Yaskawa INFORM job: DPRINT3D14.JBI

/JOB
//NAME DPRINT3D14
//POS
///NPOS 1103,0,0,0,0,0
///TOOL 9
///POSTYPE PULSE
///PULSE
C00000=35589,48234,-113777,79423,-119050,-86602,0
C00001=36149,47910,-114639,78756,-119195,-86909,0
C00002=39346,46465,-118547,75010,-120071,-88397,0
C00003=40415,47046,-117012,74132,-121018,-88120,0
C00004=36113,47361,-116093,78604,-118868,-87310,0
C00005=40186,44054,-125164,73265,-118809,-90339,0
C00006=40186,43993,-125176,73276,-118834,-90313,0
C00007=35105,44450,-123810,78705,-116693,-89341,0
C00008=36407,44998,-122328,77544,-117679,-89063,0
C00009=36336,47795,-114813,78560,-119287,-86953,0
C00010=40997,44020,-125117,72434,-119231,-90399,0
C00011=39991,43550,-126414,73325,-118416,-90634,0
C00012=35373,47318,-116057,79359,-118479,-87184,0
C00013=36258,47755,-114917,78624,-119220,-86972,0
C00014=35643,48123,-113935,79362,-119070,-86625,0
C00015=36516,48577,-112760,78655,-119824,-86406,0
C00016=42226,43977,-125263,71121,-119762,-90600,0
C00017=39858,42875,-128320,73230,-117847,-91152,0
C00018=34271,47458,-115667,80501,-117931,-86950,0
C00019=35173,47889,-114544,79748,-118673,-86739,0
C00020=34938,48134,-113895,80062,-118666,-86531,0
C00021=35406,48369,-113288,79679,-119063,-86417,0
C00022=35589,48179,-113789,79434,-119069,-86578,0
C00023=36149,47855,-114651,78767,-119213,-86885,0
C00024=39346,46408,-118558,75022,-120093,-88372,0
C00025=40382,46970,-117074,74172,-121010,-88104,0
C00026=36113,47305,-116105,78615,-118886,-87285,0
C00027=40186,43993,-125176,73276,-118834,-90313,0
C00028=40187,43932,-125189,73288,-118859,-90287,0
C00029=35144,44406,-123780,78681,-116742,-89307,0
C00030=36408,44938,-122340,77555,-117701,-89037,0
C00031=36336,47739,-114825,78571,-119305,-86929,0
C00032=40998,43959,-125128,72446,-119256,-90373,0
C00033=39991,43488,-126425,73337,-118441,-90607,0
C00034=35373,47262,-116069,79370,-118497,-87160,0
C00035=36259,47699,-114928,78635,-119239,-86948,0
C00036=35643,48068,-113947,79373,-119088,-86601,0
C00037=36517,48522,-112772,78666,-119842,-86382,0
C00038=42227,43916,-125274,71133,-119788,-90574,0
C00039=39859,42812,-128333,73241,-117873,-91125,0
C00040=34271,47402,-115679,80511,-117948,-86926,0
C00041=35173,47834,-114556,79759,-118692,-86714,0
C00042=34938,48079,-113907,80073,-118685,-86507,0
C00043=35406,48314,-113299,79690,-119081,-86392,0
C00044=35589,48124,-113800,79445,-119086,-86554,0
C00045=36150,47799,-114663,78778,-119233,-86861,0
C00046=39347,46350,-118571,75034,-120114,-88347,0
C00047=40348,46895,-117136,74211,-121001,-88089,0
C00048=36114,47249,-116118,78626,-118905,-87261,0
C00049=40187,43932,-125189,73288,-118859,-90287,0
C00050=40187,43871,-125200,73300,-118885,-90260,0
C00051=35183,44361,-123750,78656,-116791,-89272,0
C00052=36408,44879,-122352,77566,-117722,-89011,0
C00053=36337,47684,-114837,78583,-119324,-86904,0
C00054=40998,43898,-125141,72457,-119282,-90347,0
C00055=39992,43426,-126438,73348,-118466,-90581,0
C00056=35373,47206,-116081,79381,-118516,-87135,0
C00057=36259,47644,-114940,78647,-119258,-86923,0
C00058=35643,48013,-113959,79384,-119105,-86577,0
C00059=36517,48468,-112784,78678,-119860,-86358,0
C00060=42227,43855,-125287,71145,-119816,-90548,0
C00061=39859,42749,-128346,73252,-117899,-91098,0
C00062=34272,47346,-115691,80521,-117965,-86901,0
C00063=35174,47778,-114567,79770,-118709,-86690,0
C00064=34938,48024,-113919,80084,-118702,-86482,0
C00065=35407,48259,-113311,79701,-119098,-86369,0
C00066=35589,48069,-113812,79456,-119104,-86529,0
C00067=36150,47744,-114675,78789,-119251,-86836,0
C00068=39347,46293,-118583,75046,-120136,-88322,0
C00069=40315,46819,-117198,74251,-120993,-88073,0
C00070=36114,47193,-116129,78637,-118924,-87236,0
C00071=40187,43871,-125200,73300,-118885,-90260,0
C00072=40188,43810,-125213,73311,-118909,-90234,0
C00073=35222,44317,-123719,78632,-116840,-89237,0
C00074=36408,44820,-122364,77576,-117742,-88985,0
C00075=36337,47628,-114848,78594,-119343,-86880,0
C00076=40999,43837,-125153,72469,-119308,-90321,0
C00077=39992,43364,-126451,73360,-118492,-90554,0
C00078=35374,47150,-116092,79391,-118534,-87111,0
C00079=36259,47588,-114951,78658,-119277,-86899,0
C00080=35644,47958,-113971,79395,-119124,-86553,0
C00081=36517,48413,-112796,78689,-119879,-86334,0
C00082=42228,43794,-125299,71157,-119842,-90523,0
C00083=39860,42686,-128357,73264,-117925,-91071,0
C00084=34272,47291,-115703,80532,-117984,-86876,0
C00085=35174,47723,-114579,79780,-118727,-86666,0
C00086=34938,47969,-113930,80095,-118719,-86458,0
C00087=35407,48204,-113323,79712,-119117,-86344,0
C00088=35590,48014,-113824,79467,-119123,-86505,0
C00089=36150,47688,-114686,78800,-119270,-86812,0
C00090=39347,46236,-118594,75058,-120158,-88298,0
C00091=40282,46743,-117259,74291,-120985,-88058,0
C00092=36114,47136,-116141,78648,-118943,-87212,0
C00093=40188,43810,-125213,73311,-118909,-90234,0
C00094=40188,43749,-125225,73323,-118934,-90208,0
C00095=35261,44273,-123689,78608,-116890,-89203,0
C00096=36409,44760,-122376,77587,-117764,-88960,0
C00097=36337,47573,-114860,78605,-119362,-86855,0
C00098=40999,43776,-125165,72481,-119333,-90295,0
C00099=39992,43303,-126462,73371,-118517,-90527,0
C00100=35374,47094,-116104,79402,-118553,-87086,0
C00101=36259,47533,-114963,78669,-119295,-86875,0
C00102=35644,47903,-113982,79406,-119142,-86528,0
C00103=36518,48359,-112807,78701,-119897,-86310,0
C00104=42228,43733,-125311,71169,-119868,-90497,0
C00105=39860,42623,-128370,73275,-117950,-91044,0
C00106=34272,47235,-115714,80542,-118001,-86851,0
C00107=35174,47668,-114591,79791,-118746,-86641,0
C00108=34939,47914,-113942,80106,-118738,-86434,0
C00109=35407,48149,-113334,79723,-119134,-86320,0
C00110=35590,47959,-113835,79478,-119140,-86481,0
C00111=36151,47633,-114698,78812,-119288,-86788,0
C00112=39348,46179,-118605,75070,-120181,-88273,0
C00113=40248,46668,-117320,74331,-120977,-88042,0
C00114=36114,47080,-116152,78659,-118962,-87187,0
C00115=40188,43749,-125225,73323,-118934,-90208,0
C00116=40188,43688,-125237,73335,-118959,-90182,0
C00117=35300,44228,-123658,78583,-116939,-89168,0
C00118=36409,44701,-122387,77598,-117785,-88933,0
C00119=36338,47517,-114872,78617,-119381,-86831,0
C00120=40999,43715,-125178,72493,-119359,-90269,0
C00121=39993,43241,-126475,73383,-118542,-90501,0
C00122=35374,47038,-116115,79413,-118571,-87061,0
C00123=36260,47477,-114974,78680,-119315,-86850,0
C00124=35645,47848,-113994,79417,-119161,-86504,0
C00125=36518,48304,-112819,78712,-119916,-86286,0
C00126=42228,43672,-125323,71182,-119895,-90471,0
C00127=39861,42560,-128383,73286,-117977,-91017,0
C00128=34273,47179,-115726,80553,-118018,-86826,0
C00129=35175,47612,-114602,79802,-118763,-86617,0
C00130=34939,47859,-113953,80116,-118755,-86409,0
C00131=35408,48095,-113346,79734,-119151,-86296,0
C00132=35590,47904,-113847,79489,-119158,-86456,0
C00133=36151,47578,-114710,78823,-119306,-86763,0
C00134=39348,46121,-118618,75082,-120203,-88248,0
C00135=40215,46592,-117382,74371,-120969,-88026,0
C00136=36115,47024,-116165,78670,-118981,-87162,0
C00137=40188,43688,-125237,73335,-118959,-90182,0
C00138=40189,43627,-125249,73347,-118985,-90155,0
C00139=35338,44184,-123627,78559,-116989,-89134,0
C00140=36409,44642,-122400,77609,-117807,-88907,0
C00141=36338,47462,-114883,78628,-119400,-86806,0
C00142=41000,43655,-125189,72505,-119385,-90242,0
C00143=39993,43179,-126486,73394,-118568,-90475,0
C00144=35375,46982,-116127,79424,-118589,-87036,0
C00145=36260,47422,-114986,78692,-119333,-86825,0
C00146=35645,47793,-114005,79428,-119178,-86479,0
C00147=36519,48250,-112830,78724,-119934,-86262,0
C00148=42229,43611,-125335,71194,-119922,-90445,0
C00149=39861,42497,-128394,73298,-118003,-90990,0
C00150=34273,47123,-115737,80563,-118037,-86802,0
C00151=35175,47557,-114614,79813,-118781,-86592,0
C00152=34939,47804,-113965,80127,-118772,-86384,0
C00153=35408,48040,-113357,79745,-119170,-86272,0
C00154=35591,47849,-113858,79501,-119177,-86432,0
C00155=36151,47522,-114721,78834,-119326,-86739,0
C00156=39349,46064,-118630,75094,-120225,-88223,0
C00157=40181,46517,-117443,74411,-120961,-88011,0
C00158=36115,46968,-116176,78681,-119000,-87137,0
C00159=40189,43627,-125249,73347,-118985,-90155,0
C00160=40189,43566,-125261,73358,-119010,-90129,0
C00161=35377,44140,-123596,78535,-117038,-89099,0
C00162=36410,44583,-122411,77620,-117828,-88881,0
C00163=36338,47406,-114894,78639,-119418,-86782,0
C00164=41000,43594,-125200,72517,-119411,-90216,0
C00165=39994,43117,-126499,73406,-118593,-90448,0
C00166=35375,46926,-116138,79435,-118608,-87011,0
C00167=36260,47366,-114997,78703,-119351,-86801,0
C00168=35645,47738,-114017,79439,-119196,-86455,0
C00169=36519,48195,-112841,78735,-119952,-86238,0
C00170=42229,43550,-125346,71206,-119949,-90419,0
C00171=39861,42434,-128407,73309,-118029,-90963,0
C00172=34273,47067,-115749,80574,-118054,-86777,0
C00173=35175,47502,-114625,79824,-118799,-86568,0
C00174=34940,47749,-113976,80138,-118791,-86360,0
C00175=35408,47985,-113369,79756,-119187,-86247,0
C00176=35591,47794,-113870,79512,-119195,-86408,0
C00177=36152,47467,-114732,78846,-119344,-86714,0
C00178=36115,46912,-116187,78693,-119019,-87113,0
C00179=40189,43566,-125261,73358,-119010,-90129,0
C00180=40190,43505,-125273,73370,-119035,-90103,0
C00181=35416,44096,-123565,78512,-117087,-89065,0
C00182=36410,44523,-122423,77631,-117848,-88854,0
C00183=36339,47351,-114906,78651,-119437,-86757,0
C00184=41001,43533,-125213,72529,-119436,-90190,0
C00185=39994,43056,-126511,73418,-118618,-90421,0
C00186=35375,46870,-116150,79446,-118626,-86986,0
C00187=36261,47311,-115009,78714,-119371,-86776,0
C00188=35646,47683,-114028,79451,-119215,-86430,0
C00189=36519,48141,-112853,78747,-119971,-86214,0
C00190=42230,43489,-125359,71219,-119975,-90393,0
C00191=39862,42371,-128418,73320,-118055,-90935,0
C00192=34274,47011,-115760,80584,-118071,-86752,0
C00193=35176,47446,-114636,79835,-118817,-86543,0
C00194=34940,47694,-113987,80149,-118808,-86336,0
C00195=35409,47930,-113380,79768,-119205,-86223,0
C00196=35591,47739,-113881,79523,-119212,-86383,0
C00197=36152,47412,-114744,78857,-119363,-86690,0
C00198=36116,46856,-116198,78704,-119039,-87088,0
C00199=40190,43505,-125273,73370,-119035,-90103,0
C00200=40190,43444,-125284,73382,-119059,-90077,0
C00201=35455,44052,-123534,78488,-117137,-89030,0
C00202=36410,44464,-122434,77642,-117870,-88828,0
C00203=36339,47296,-114917,78662,-119456,-86732,0
C00204=41001,43472,-125225,72541,-119463,-90164,0
C00205=39994,42994,-126522,73429,-118645,-90395,0
C00206=35376,46814,-116161,79457,-118646,-86961,0
C00207=36261,47256,-115020,78726,-119389,-86752,0
C00208=35646,47628,-114039,79462,-119233,-86406,0
C00209=36519,48086,-112864,78758,-119990,-86189,0
C00210=42230,43428,-125371,71231,-120003,-90367,0
C00211=39862,42308,-128431,73332,-118081,-90909,0
C00212=34274,46956,-115772,80595,-118090,-86727,0
C00213=35176,47391,-114648,79846,-118835,-86518,0
C00214=34940,47639,-113999,80160,-118825,-86311,0
C00215=35409,47876,-113391,79779,-119223,-86199,0
C00216=35592,47684,-113892,79534,-119231,-86359,0
C00217=36152,47356,-114755,78868,-119382,-86665,0
C00218=36116,46800,-116210,78715,-119057,-87063,0
C00219=40190,43444,-125284,73382,-119059,-90077,0
C00220=40190,43384,-125296,73394,-119085,-90050,0
C00221=35493,44009,-123502,78464,-117186,-88996,0
C00222=36411,44405,-122446,77653,-117891,-88802,0
C00223=36339,47240,-114928,78673,-119475,-86708,0
C00224=41001,43411,-125236,72554,-119488,-90138,0
C00225=39995,42932,-126534,73441,-118670,-90368,0
C00226=35376,46758,-116173,79468,-118664,-86936,0
C00227=36261,47200,-115032,78737,-119409,-86727,0
C00228=35646,47573,-114050,79473,-119251,-86381,0
C00229=36520,48032,-112875,78770,-120009,-86166,0
C00230=42231,43367,-125382,71244,-120029,-90341,0
C00231=39863,42246,-128442,73343,-118107,-90881,0
C00232=34274,46900,-115782,80606,-118107,-86702,0
C00233=35176,47336,-114659,79857,-118853,-86493,0
C00234=34941,47584,-114010,80171,-118843,-86286,0
C00235=35409,47821,-113402,79790,-119241,-86174,0
C00236=35592,47629,-113903,79545,-119249,-86334,0
C00237=36153,47301,-114766,78880,-119401,-86640,0
C00238=36116,46744,-116221,78726,-119077,-87038,0
C00239=40190,43384,-125296,73394,-119085,-90050,0
C00240=40191,43323,-125307,73406,-119110,-90024,0
C00241=36340,47185,-114939,78685,-119494,-86683,0
C00242=41002,43350,-125248,72566,-119513,-90111,0
C00243=39995,42871,-126546,73453,-118695,-90341,0
C00244=35376,46702,-116183,79479,-118682,-86911,0
C00245=36262,47145,-115042,78749,-119427,-86702,0
C00246=35646,47518,-114061,79484,-119270,-86357,0
C00247=36520,47977,-112886,78782,-120027,-86141,0
C00248=42231,43306,-125394,71256,-120056,-90314,0
C00249=39863,42183,-128454,73355,-118133,-90854,0
C00250=34275,46844,-115794,80616,-118124,-86677,0
C00251=35177,47281,-114670,79868,-118871,-86469,0
C00252=34941,47529,-114021,80182,-118861,-86262,0
C00253=35410,47766,-113413,79801,-119259,-86150,0
C00254=35592,47574,-113914,79557,-119267,-86310,0
C00255=36153,47246,-114777,78891,-119419,-86616,0
C00256=36117,46688,-116231,78738,-119095,-87013,0
C00257=40191,43323,-125307,73406,-119110,-90024,0
C00258=40191,43262,-125319,73418,-119135,-89997,0
C00259=36340,47130,-114950,78696,-119513,-86659,0
C00260=41002,43290,-125259,72578,-119540,-90085,0
C00261=39996,42809,-126558,73465,-118720,-90314,0
C00262=35377,46646,-116195,79490,-118701,-86886,0
C00263=36262,47090,-115053,78760,-119447,-86677,0
C00264=35647,47463,-114072,79496,-119287,-86332,0
C00265=36520,47923,-112897,78793,-120045,-86117,0
C00266=42231,43245,-125405,71269,-120083,-90288,0
C00267=39864,42120,-128465,73367,-118160,-90827,0
C00268=34275,46789,-115804,80627,-118142,-86652,0
C00269=35177,47226,-114681,79879,-118889,-86444,0
C00270=34941,47474,-114032,80193,-118878,-86237,0
C00271=35410,47712,-113424,79812,-119277,-86125,0
C00272=35593,47519,-113925,79568,-119285,-86285,0
C00273=36153,47191,-114788,78903,-119439,-86591,0
C00274=36117,46633,-116243,78749,-119115,-86988,0
C00275=40191,43262,-125319,73418,-119135,-89997,0
C00276=40192,43201,-125330,73430,-119161,-89971,0
C00277=36340,47074,-114960,78708,-119532,-86634,0
C00278=41003,43229,-125271,72590,-119565,-90059,0
C00279=39996,42748,-126569,73476,-118746,-90287,0
C00280=35377,46590,-116205,79501,-118719,-86861,0
C00281=36263,47034,-115064,78772,-119465,-86653,0
C00282=35647,47408,-114083,79507,-119305,-86308,0
C00283=36521,47869,-112908,78805,-120064,-86092,0
C00284=42232,43185,-125417,71281,-120110,-90262,0
C00285=39864,42057,-128477,73378,-118186,-90799,0
C00286=34275,46733,-115815,80638,-118160,-86627,0
C00287=35177,47171,-114692,79890,-118907,-86420,0
C00288=34942,47419,-114042,80204,-118896,-86213,0
C00289=35410,47657,-113435,79824,-119295,-86101,0
C00290=35593,47465,-113936,79579,-119303,-86261,0
C00291=36154,47136,-114799,78914,-119457,-86567,0
C00292=36118,46577,-116254,78760,-119134,-86963,0
C00293=40192,43201,-125330,73430,-119161,-89971,0
C00294=40192,43140,-125342,73442,-119186,-89944,0
C00295=36341,47019,-114972,78720,-119551,-86609,0
C00296=41003,43168,-125281,72602,-119591,-90032,0
C00297=39997,42686,-126579,73488,-118772,-90260,0
C00298=35377,46535,-116216,79512,-118738,-86836,0
C00299=36263,46979,-115075,78783,-119485,-86628,0
C00300=35647,47353,-114094,79518,-119324,-86283,0
C00301=36521,47815,-112918,78817,-120082,-86068,0
C00302=42232,43124,-125427,71294,-120137,-90236,0
C00303=39864,41994,-128488,73390,-118211,-90772,0
C00304=34276,46677,-115826,80649,-118178,-86601,0
C00305=35177,47115,-114702,79902,-118925,-86395,0
C00306=34942,47365,-114053,80215,-118913,-86188,0
C00307=35411,47603,-113446,79835,-119312,-86076,0
C00308=35593,47410,-113947,79591,-119321,-86236,0
C00309=36154,47080,-114810,78925,-119475,-86542,0
C00310=36118,46521,-116265,78772,-119152,-86938,0
C00311=40192,43140,-125342,73442,-119186,-89944,0
C00312=40192,43080,-125352,73454,-119211,-89918,0
C00313=36341,46964,-114982,78731,-119570,-86584,0
C00314=41003,43108,-125292,72615,-119617,-90006,0
C00315=39997,42625,-126591,73500,-118797,-90234,0
C00316=35378,46479,-116227,79524,-118757,-86811,0
C00317=36263,46924,-115086,78795,-119503,-86603,0
C00318=35648,47299,-114104,79530,-119342,-86258,0
C00319=36521,47760,-112929,78829,-120101,-86044,0
C00320=42233,43063,-125438,71306,-120164,-90210,0
C00321=39865,41932,-128500,73402,-118238,-90744,0
C00322=34276,46622,-115837,80659,-118195,-86576,0
C00323=35178,47060,-114713,79913,-118943,-86370,0
C00324=34942,47310,-114064,80226,-118932,-86163,0
C00325=35411,47548,-113456,79846,-119331,-86052,0
C00326=35594,47355,-113958,79602,-119340,-86211,0
C00327=36154,47025,-114820,78937,-119495,-86517,0
C00328=36118,46465,-116275,78783,-119172,-86913,0
C00329=40192,43080,-125352,73454,-119211,-89918,0
C00330=40193,43019,-125364,73466,-119236,-89891,0
C00331=36341,46909,-114993,78743,-119589,-86560,0
C00332=41004,43047,-125304,72627,-119643,-89980,0
C00333=39997,42563,-126602,73512,-118823,-90207,0
C00334=35378,46423,-116237,79535,-118776,-86786,0
C00335=36264,46868,-115096,78806,-119521,-86579,0
C00336=35648,47244,-114115,79541,-119360,-86234,0
C00337=36522,47706,-112940,78840,-120119,-86019,0
C00338=42233,43002,-125450,71319,-120191,-90184,0
C00339=39865,41869,-128511,73413,-118264,-90717,0
C00340=34276,46566,-115848,80670,-118212,-86551,0
C00341=35178,47005,-114724,79924,-118962,-86345,0
C00342=34943,47255,-114074,80238,-118949,-86138,0
C00343=35411,47494,-113467,79858,-119348,-86027,0
C00344=35594,47301,-113968,79613,-119357,-86187,0
C00345=36155,46970,-114831,78948,-119513,-86492,0
C00346=36119,46409,-116286,78795,-119192,-86888,0
C00347=40193,43019,-125364,73466,-119236,-89891,0
C00348=40193,42958,-125375,73478,-119262,-89865,0
C00349=36342,46854,-115004,78754,-119608,-86535,0
C00350=41004,42986,-125314,72640,-119670,-89954,0
C00351=39998,42502,-126613,73524,-118848,-90180,0
C00352=35378,46367,-116249,79546,-118794,-86761,0
C00353=36264,46813,-115106,78818,-119541,-86554,0
C00354=35648,47189,-114126,79552,-119379,-86209,0
C00355=36522,47652,-112950,78852,-120137,-85995,0
C00356=42234,42942,-125460,71332,-120218,-90157,0
C00357=39866,41806,-128523,73425,-118291,-90689,0
C00358=34276,46511,-115858,80681,-118231,-86526,0
C00359=35178,46950,-114734,79935,-118979,-86320,0
C00360=34943,47200,-114085,80249,-118967,-86114,0
C00361=35412,47439,-113477,79869,-119366,-86002,0
C00362=35594,47246,-113979,79625,-119375,-86162,0
C00363=36155,46915,-114842,78960,-119532,-86467,0
C00364=36119,46354,-116297,78806,-119210,-86862,0
C00365=40193,42958,-125375,73478,-119262,-89865,0
C00366=40194,42898,-125386,73490,-119287,-89838,0
C00367=36342,46799,-115014,78766,-119627,-86510,0
C00368=41005,42926,-125326,72652,-119695,-89927,0
C00369=39998,42440,-126624,73536,-118874,-90153,0
C00370=35379,46312,-116259,79557,-118812,-86735,0
C00371=36264,46758,-115118,78829,-119559,-86529,0
C00372=35649,47135,-114136,79564,-119397,-86184,0
C00373=36522,47598,-112960,78864,-120157,-85971,0
C00374=42234,42881,-125472,71345,-120245,-90131,0
C00375=39866,41744,-128533,73437,-118317,-90662,0
C00376=34277,46455,-115868,80692,-118248,-86501,0
C00377=35179,46895,-114745,79947,-118997,-86296,0
C00378=34943,47146,-114096,80260,-118985,-86089,0
C00379=35412,47385,-113488,79880,-119383,-85978,0
C00380=35595,47191,-113989,79636,-119394,-86138,0
C00381=36155,46860,-114852,78972,-119551,-86442,0
C00382=36119,46298,-116307,78818,-119229,-86837,0
C00383=40194,42898,-125386,73490,-119287,-89838,0
C00384=40194,42837,-125397,73503,-119312,-89811,0
C00385=36342,46744,-115025,78778,-119645,-86485,0
C00386=41005,42865,-125336,72664,-119721,-89900,0
C00387=39999,42379,-126636,73548,-118900,-90126,0
C00388=35379,46256,-116269,79569,-118831,-86710,0
C00389=36265,46703,-115128,78841,-119579,-86504,0
C00390=35649,47080,-114146,79575,-119414,-86160,0
C00391=36523,47544,-112971,78876,-120175,-85946,0
C00392=42234,42820,-125482,71357,-120272,-90105,0
C00393=39866,41681,-128545,73449,-118343,-90635,0
C00394=34277,46400,-115879,80703,-118266,-86475,0
C00395=35179,46840,-114755,79958,-119016,-86271,0
C00396=34944,47091,-114106,80271,-119002,-86064,0
C00397=35412,47331,-113498,79892,-119402,-85953,0
C00398=35595,47137,-114000,79648,-119412,-86113,0
C00399=36156,46805,-114862,78983,-119570,-86418,0
C00400=41102,41865,-128063,72210,-119040,-90656,0
C00401=41544,42076,-127493,71817,-119398,-90558,0
C00402=35038,47556,-112914,80333,-119290,-85748,0
C00403=34622,47344,-113451,80668,-118935,-85846,0
C00404=36120,46242,-116318,78829,-119249,-86813,0
C00405=40194,42837,-125397,73503,-119312,-89811,0
C00406=40194,42776,-125407,73515,-119338,-89785,0
C00407=36343,46688,-115035,78790,-119665,-86460,0
C00408=41005,42805,-125348,72677,-119747,-89873,0
C00409=39999,42318,-126646,73560,-118925,-90099,0
C00410=35379,46200,-116280,79580,-118850,-86685,0
C00411=36265,46648,-115138,78853,-119598,-86479,0
C00412=35649,47025,-114157,79587,-119433,-86135,0
C00413=36523,47489,-112981,78888,-120194,-85922,0
C00414=42235,42760,-125494,71370,-120299,-90078,0
C00415=39867,41618,-128555,73460,-118369,-90607,0
C00416=34277,46344,-115889,80713,-118284,-86450,0
C00417=35179,46785,-114765,79969,-119034,-86246,0
C00418=34944,47036,-114116,80282,-119020,-86039,0
C00419=35412,47276,-113508,79903,-119420,-85928,0
C00420=35595,47082,-114010,79659,-119431,-86088,0
C00421=36156,46750,-114873,78995,-119588,-86393,0
C00422=41093,41808,-128058,72234,-119066,-90623,0
C00423=41536,42020,-127488,71841,-119426,-90525,0
C00424=35045,47495,-112943,80335,-119308,-85729,0
C00425=34629,47282,-113480,80671,-118953,-85828,0
C00426=36120,46186,-116328,78841,-119269,-86787,0
C00427=40194,42776,-125407,73515,-119338,-89785,0
C00428=40195,42716,-125418,73527,-119363,-89758,0
C00429=36343,46633,-115045,78801,-119683,-86435,0
C00430=41006,42744,-125358,72689,-119773,-89847,0
C00431=39999,42256,-126656,73572,-118951,-90071,0
C00432=35380,46145,-116290,79591,-118869,-86660,0
C00433=36265,46593,-115148,78865,-119617,-86454,0
C00434=35650,46971,-114167,79598,-119451,-86110,0
C00435=36523,47435,-112991,78900,-120212,-85897,0
C00436=42235,42699,-125504,71383,-120326,-90052,0
C00437=39867,41556,-128566,73472,-118395,-90579,0
C00438=34278,46289,-115899,80724,-118302,-86425,0
C00439=35180,46731,-114776,79980,-119051,-86221,0
C00440=34944,46982,-114126,80294,-119038,-86014,0
C00441=35413,47222,-113519,79915,-119437,-85904,0
C00442=35596,47028,-114020,79671,-119449,-86063,0
C00443=36156,46695,-114883,79007,-119608,-86368,0
C00444=36120,46131,-116338,78852,-119287,-86762,0
C00445=40195,42716,-125418,73527,-119363,-89758,0
C00446=40195,42655,-125428,73540,-119388,-89731,0
C00447=36344,46578,-115055,78813,-119703,-86410,0
C00448=41006,42683,-125368,72702,-119799,-89821,0
C00449=40000,42195,-126668,73584,-118977,-90045,0
C00450=35380,46089,-116300,79602,-118887,-86634,0
C00451=36265,46538,-115158,78876,-119636,-86429,0
C00452=35650,46916,-114177,79610,-119470,-86085,0
C00453=36524,47381,-113001,78912,-120230,-85873,0
C00454=42236,42638,-125514,71396,-120353,-90025,0
C00455=39868,41493,-128577,73484,-118422,-90552,0
C00456=34278,46233,-115910,80735,-118319,-86400,0
C00457=35180,46676,-114786,79992,-119070,-86195,0
C00458=34945,46927,-114136,80305,-119056,-85989,0
C00459=35413,47168,-113529,79926,-119456,-85879,0
C00460=35596,46973,-114030,79682,-119466,-86038,0
C00461=36157,46640,-114893,79018,-119626,-86343,0
C00462=36121,46075,-116349,78864,-119306,-86737,0
C00463=40195,42655,-125428,73540,-119388,-89731,0
C00464=40196,42595,-125438,73552,-119413,-89704,0
C00465=36344,46523,-115065,78825,-119721,-86385,0
C00466=41007,42623,-125379,72715,-119825,-89794,0
C00467=40000,42134,-126678,73597,-119002,-90017,0
C00468=35380,46034,-116309,79614,-118905,-86609,0
C00469=36266,46483,-115168,78888,-119655,-86404,0
C00470=35650,46861,-114187,79622,-119488,-86060,0
C00471=36524,47327,-113011,78924,-120250,-85848,0
C00472=42236,42578,-125525,71409,-120380,-89999,0
C00473=39868,41431,-128588,73496,-118448,-90524,0
C00474=34278,46178,-115920,80746,-118337,-86374,0
C00475=35180,46621,-114796,80003,-119088,-86170,0
C00476=34945,46873,-114147,80316,-119073,-85965,0
C00477=35414,47113,-113539,79938,-119474,-85854,0
C00478=35596,46918,-114040,79694,-119485,-86014,0
C00479=36157,46585,-114903,79030,-119645,-86318,0
C00480=36121,46020,-116359,78876,-119326,-86712,0
C00481=40196,42595,-125438,73552,-119413,-89704,0
C00482=40196,42534,-125450,73564,-119439,-89677,0
C00483=36344,46469,-115075,78837,-119741,-86361,0
C00484=41007,42562,-125389,72727,-119851,-89767,0
C00485=40001,42072,-126689,73609,-119028,-89990,0
C00486=35381,45978,-116320,79625,-118925,-86584,0
C00487=36266,46428,-115179,78900,-119674,-86379,0
C00488=35651,46807,-114197,79633,-119506,-86035,0
C00489=36524,47273,-113021,78936,-120268,-85823,0
C00490=42237,42517,-125535,71422,-120407,-89973,0
C00491=39869,41368,-128599,73508,-118474,-90496,0
C00492=34279,46123,-115930,80757,-118355,-86349,0
C00493=35181,46566,-114806,80015,-119107,-86145,0
C00494=34945,46818,-114156,80328,-119092,-85939,0
C00495=35414,47059,-113549,79950,-119491,-85830,0
C00496=35597,46864,-114050,79705,-119503,-85989,0
C00497=36157,46531,-114913,79042,-119664,-86293,0
C00498=36121,45964,-116368,78887,-119346,-86686,0
C00499=40196,42534,-125450,73564,-119439,-89677,0
C00500=40197,42474,-125459,73577,-119465,-89651,0
C00501=36344,46414,-115084,78849,-119760,-86335,0
C00502=41008,42502,-125399,72740,-119876,-89741,0
C00503=40001,42011,-126699,73621,-119054,-89963,0
C00504=35381,45923,-116330,79637,-118943,-86558,0
C00505=36266,46373,-115188,78912,-119693,-86354,0
C00506=35651,46752,-114207,79645,-119525,-86011,0
C00507=36525,47219,-113031,78948,-120287,-85799,0
C00508=42237,42457,-125545,71435,-120434,-89946,0
C00509=39869,41306,-128609,73520,-118501,-90469,0
C00510=34279,46067,-115939,80768,-118372,-86323,0
C00511=35181,46511,-114816,80026,-119124,-86120,0
C00512=34946,46764,-114166,80339,-119109,-85914,0
C00513=35414,47005,-113559,79961,-119510,-85805,0
C00514=35597,46809,-114060,79717,-119521,-85964,0
C00515=36158,46476,-114922,79054,-119682,-86268,0
C00516=39612,44893,-119069,75037,-120734,-87842,0
C00517=39283,45170,-118342,75471,-120723,-87602,0
C00518=36122,45909,-116378,78899,-119364,-86661,0
C00519=40197,42474,-125459,73577,-119465,-89651,0
C00520=40197,42413,-125469,73589,-119490,-89623,0
C00521=36345,46359,-115095,78860,-119779,-86310,0
C00522=41008,42442,-125410,72753,-119903,-89714,0
C00523=40001,41950,-126709,73633,-119079,-89936,0
C00524=35381,45867,-116339,79648,-118962,-86533,0
C00525=36267,46318,-115198,78924,-119712,-86329,0
C00526=35651,46698,-114217,79657,-119543,-85985,0
C00527=36525,47165,-113041,78960,-120305,-85774,0
C00528=42237,42396,-125556,71448,-120461,-89919,0
C00529=39869,41243,-128619,73532,-118527,-90441,0
C00530=34279,46012,-115950,80779,-118391,-86298,0
C00531=35181,46457,-114825,80037,-119142,-86095,0
C00532=34946,46709,-114176,80350,-119127,-85889,0
C00533=35414,46951,-113568,79973,-119528,-85780,0
C00534=35597,46755,-114070,79729,-119540,-85939,0
C00535=36158,46421,-114933,79066,-119702,-86243,0
C00536=36122,45853,-116389,78911,-119383,-86636,0
C00537=40197,42413,-125469,73589,-119490,-89623,0
C00538=40197,42353,-125480,73602,-119516,-89597,0
C00539=36345,46304,-115104,78872,-119798,-86285,0
C00540=41008,42381,-125420,72765,-119929,-89687,0
C00541=40002,41889,-126720,73646,-119105,-89908,0
C00542=35382,45812,-116350,79660,-118981,-86507,0
C00543=36267,46263,-115207,78935,-119731,-86304,0
C00544=35652,46643,-114226,79668,-119562,-85960,0
C00545=36525,47111,-113051,78972,-120323,-85749,0
C00546=42238,42336,-125566,71461,-120489,-89893,0
C00547=39870,41181,-128630,73544,-118554,-90413,0
C00548=34280,45957,-115959,80790,-118408,-86273,0
C00549=35182,46402,-114835,80049,-119161,-86070,0
C00550=34946,46655,-114186,80362,-119144,-85864,0
C00551=35415,46897,-113578,79984,-119546,-85755,0
C00552=35598,46701,-114079,79740,-119558,-85914,0
C00553=36158,46366,-114942,79077,-119720,-86218,0
C00554=36122,45798,-116398,78923,-119403,-86610,0
C00555=40197,42353,-125480,73602,-119516,-89597,0
C00556=40198,42293,-125490,73614,-119541,-89570,0
C00557=36345,46249,-115114,78884,-119817,-86260,0
C00558=41009,42321,-125430,72778,-119956,-89660,0
C00559=40002,41828,-126730,73658,-119131,-89881,0
C00560=35382,45756,-116359,79671,-119000,-86482,0
C00561=36268,46208,-115218,78947,-119750,-86278,0
C00562=35652,46589,-114236,79680,-119580,-85935,0
C00563=36526,47057,-113060,78984,-120343,-85725,0
C00564=42238,42275,-125576,71474,-120515,-89866,0
C00565=39870,41118,-128640,73557,-118580,-90385,0
C00566=34280,45902,-115969,80801,-118426,-86247,0
C00567=35182,46347,-114845,80060,-119179,-86045,0
C00568=34947,46600,-114195,80373,-119163,-85839,0
C00569=35415,46842,-113588,79996,-119564,-85730,0
C00570=35598,46646,-114089,79752,-119577,-85889,0
C00571=36159,46311,-114952,79089,-119740,-86193,0
C00572=36123,45742,-116408,78934,-119423,-86584,0
C00573=40198,42293,-125490,73614,-119541,-89570,0
C00574=40198,42232,-125500,73627,-119566,-89543,0
C00575=36479,43102,-123131,77745,-118223,-88438,0
C00576=36161,43380,-122393,78158,-118212,-88198,0
C00577=36346,46194,-115124,78896,-119836,-86235,0
C00578=41009,42261,-125440,72791,-119981,-89633,0
C00579=40003,41767,-126739,73671,-119157,-89854,0
C00580=35382,45701,-116369,79683,-119018,-86457,0
C00581=36268,46153,-115227,78959,-119770,-86253,0
C00582=35652,46535,-114246,79692,-119598,-85910,0
C00583=36526,47004,-113070,78996,-120361,-85700,0
C00584=42239,42215,-125585,71487,-120543,-89839,0
C00585=39871,41056,-128650,73569,-118607,-90357,0
C00586=34280,45846,-115979,80813,-118443,-86222,0
C00587=35182,46292,-114854,80072,-119197,-86019,0
C00588=34946,46547,-114203,80386,-119180,-85814,0
C00589=35415,46789,-113596,80008,-119582,-85705,0
C00590=35598,46592,-114099,79764,-119595,-85864,0
C00591=36159,46256,-114962,79101,-119758,-86167,0
C00592=36123,45687,-116418,78946,-119441,-86559,0
C00593=40198,42232,-125500,73627,-119566,-89543,0
C00594=40199,42172,-125510,73639,-119591,-89515,0
C00595=36346,46139,-115133,78908,-119856,-86210,0
C00596=41010,42200,-125450,72804,-120007,-89607,0
C00597=40003,41705,-126750,73683,-119182,-89826,0
C00598=35383,45646,-116378,79694,-119036,-86431,0
C00599=36268,46098,-115236,78971,-119788,-86228,0
C00600=35653,46480,-114255,79704,-119617,-85885,0
C00601=36526,46950,-113079,79009,-120380,-85675,0
C00602=42239,42154,-125596,71500,-120571,-89813,0
C00603=39871,40994,-128659,73581,-118633,-90330,0
C00604=34281,45791,-115988,80824,-118462,-86196,0
C00605=35183,46238,-114864,80084,-119216,-85994,0
C00606=34947,46492,-114214,80396,-119198,-85789,0
C00607=35416,46734,-113607,80019,-119600,-85680,0
C00608=35599,46538,-114108,79776,-119613,-85839,0
C00609=36159,46202,-114971,79113,-119778,-86142,0
C00610=36123,45631,-116427,78958,-119460,-86533,0
C00611=40199,42172,-125510,73639,-119591,-89515,0
C00612=40199,42111,-125520,73652,-119618,-89489,0
C00613=36346,46085,-115143,78920,-119874,-86184,0
C00614=41010,42140,-125460,72817,-120034,-89579,0
C00615=40003,41644,-126759,73695,-119209,-89799,0
C00616=35383,45590,-116388,79706,-119056,-86406,0
C00617=36269,46044,-115247,78983,-119808,-86203,0
C00618=35653,46426,-114264,79715,-119635,-85860,0
C00619=36527,46896,-113089,79021,-120398,-85650,0
C00620=42239,42094,-125606,71514,-120597,-89786,0
C00621=39871,40931,-128670,73593,-118660,-90302,0
C00622=34281,45736,-115998,80835,-118479,-86171,0
C00623=35183,46183,-114873,80095,-119233,-85969,0
C00624=34947,46437,-114224,80408,-119217,-85764,0
C00625=35416,46680,-113616,80031,-119618,-85655,0
C00626=35599,46483,-114117,79787,-119632,-85813,0
C00627=36160,46147,-114981,79125,-119796,-86117,0
C00628=36124,45576,-116436,78970,-119480,-86508,0
C00629=40199,42111,-125520,73652,-119618,-89489,0
C00630=40199,42051,-125529,73665,-119643,-89461,0
C00631=36347,46030,-115152,78932,-119894,-86159,0
C00632=41010,42080,-125469,72830,-120060,-89553,0
C00633=40004,41583,-126769,73708,-119234,-89771,0
C00634=35383,45535,-116397,79717,-119074,-86380,0
C00635=36269,45989,-115256,78995,-119826,-86177,0
C00636=35653,46372,-114274,79727,-119654,-85835,0
C00637=36527,46842,-113098,79033,-120418,-85625,0
C00638=42240,42034,-125615,71527,-120625,-89759,0
C00639=39872,40869,-128680,73606,-118686,-90274,0
C00640=34281,45681,-116007,80846,-118497,-86145,0
C00641=35183,46128,-114883,80107,-119251,-85944,0
C00642=34948,46383,-114233,80419,-119234,-85739,0
C00643=35416,46626,-113625,80043,-119636,-85630,0
C00644=35599,46429,-114127,79799,-119650,-85788,0
C00645=36160,46093,-114990,79137,-119816,-86092,0
C00646=36124,45521,-116446,78982,-119500,-86482,0
C00647=40199,42051,-125529,73665,-119643,-89461,0
C00648=40200,41991,-125539,73677,-119668,-89434,0
C00649=36347,45975,-115161,78945,-119913,-86134,0
C00650=41011,42020,-125479,72843,-120086,-89525,0
C00651=40004,41522,-126778,73721,-119261,-89744,0
C00652=35384,45480,-116406,79729,-119093,-86354,0
C00653=36269,45934,-115265,79007,-119845,-86152,0
C00654=35654,46317,-114283,79739,-119672,-85810,0
C00655=36527,46788,-113107,79045,-120436,-85601,0
C00656=42240,41973,-125625,71540,-120652,-89732,0
C00657=39872,40807,-128689,73618,-118712,-90245,0
C00658=34282,45626,-116016,80857,-118516,-86119,0
C00659=35184,46074,-114892,80118,-119270,-85918,0
C00660=34948,46329,-114242,80431,-119252,-85714,0
C00661=35417,46572,-113634,80055,-119654,-85605,0
C00662=35600,46375,-114136,79811,-119667,-85763,0
C00663=36160,46038,-114999,79149,-119834,-86066,0
C00664=36124,45465,-116455,78994,-119519,-86457,0
C00665=40200,41991,-125539,73677,-119668,-89434,0
C00666=40200,41931,-125549,73690,-119694,-89407,0
C00667=36347,45921,-115171,78957,-119932,-86109,0
C00668=41011,41959,-125489,72856,-120112,-89499,0
C00669=40005,41461,-126789,73733,-119286,-89717,0
C00670=35384,45424,-116415,79741,-119112,-86329,0
C00671=36270,45879,-115274,79019,-119865,-86127,0
C00672=35654,46263,-114292,79751,-119690,-85785,0
C00673=36528,46735,-113116,79058,-120454,-85576,0
C00674=42241,41913,-125635,71553,-120679,-89706,0
C00675=39873,40744,-128700,73630,-118739,-90218,0
C00676=34282,45571,-116026,80869,-118533,-86094,0
C00677=35184,46019,-114901,80130,-119288,-85893,0
C00678=34949,46274,-114251,80443,-119270,-85689,0
C00679=35417,46518,-113644,80067,-119672,-85580,0
C00680=35600,46321,-114145,79823,-119686,-85738,0
C00681=36161,45983,-115009,79161,-119853,-86041,0
C00682=36125,45410,-116465,79006,-119539,-86431,0
C00683=40200,41931,-125549,73690,-119694,-89407,0
C00684=40201,41871,-125558,73703,-119719,-89380,0
C00685=36348,45866,-115180,78969,-119951,-86083,0
C00686=41012,41899,-125498,72869,-120138,-89471,0
C00687=40005,41400,-126798,73746,-119312,-89689,0
C00688=35384,45369,-116424,79752,-119131,-86303,0
C00689=36270,45825,-115283,79032,-119883,-86101,0
C00690=35654,46209,-114301,79763,-119709,-85759,0
C00691=36528,46681,-113125,79070,-120474,-85551,0
C00692=42241,41853,-125644,71567,-120706,-89679,0
C00693=39873,40682,-128709,73643,-118765,-90190,0
C00694=34282,45516,-116035,80880,-118551,-86068,0
C00695=35184,45965,-114910,80142,-119306,-85868,0
C00696=34949,46220,-114261,80454,-119288,-85663,0
C00697=35417,46464,-113653,80078,-119690,-85555,0
C00698=35600,46267,-114154,79835,-119704,-85713,0
C00699=36161,45929,-115018,79173,-119872,-86016,0
C00700=36125,45355,-116473,79018,-119557,-86406,0
C00701=40201,41871,-125558,73703,-119719,-89380,0
C00702=40201,41810,-125567,73716,-119745,-89353,0
C00703=36348,45811,-115188,78981,-119971,-86058,0
C00704=41012,41839,-125507,72882,-120165,-89445,0
C00705=40006,41339,-126807,73758,-119338,-89662,0
C00706=35385,45314,-116434,79764,-119150,-86277,0
C00707=36270,45770,-115291,79044,-119903,-86076,0
C00708=35655,46155,-114310,79775,-119727,-85734,0
C00709=36528,46627,-113134,79082,-120492,-85526,0
C00710=42242,41793,-125653,71580,-120734,-89652,0
C00711=39874,40620,-128718,73655,-118792,-90161,0
C00712=34283,45461,-116043,80891,-118569,-86042,0
C00713=35185,45910,-114919,80153,-119325,-85842,0
C00714=34949,46166,-114270,80466,-119305,-85638,0
C00715=35418,46410,-113662,80090,-119709,-85530,0
C00716=35601,46212,-114163,79847,-119722,-85688,0
C00717=36161,45874,-115026,79185,-119891,-85991,0
C00718=36125,45300,-116482,79030,-119577,-86380,0
C00719=40201,41810,-125567,73716,-119745,-89353,0
C00720=40201,41750,-125576,73729,-119771,-89326,0
C00721=36349,45757,-115197,78993,-119989,-86033,0
C00722=41013,41779,-125517,72895,-120191,-89417,0
C00723=40006,41278,-126816,73771,-119364,-89634,0
C00724=35385,45259,-116443,79776,-119169,-86251,0
C00725=36271,45715,-115301,79056,-119922,-86051,0
C00726=35655,46100,-114319,79787,-119745,-85709,0
C00727=36529,46574,-113143,79095,-120511,-85501,0
C00728=42242,41733,-125662,71594,-120761,-89625,0
C00729=39874,40558,-128728,73668,-118818,-90133,0
C00730=34283,45406,-116052,80903,-118587,-86016,0
C00731=35185,45856,-114928,80165,-119343,-85817,0
C00732=34949,46112,-114278,80478,-119324,-85613,0
C00733=35418,46356,-113670,80102,-119726,-85505,0
C00734=35601,46158,-114172,79859,-119741,-85662,0
C00735=36162,45820,-115035,79198,-119910,-85965,0
C00736=36126,45244,-116491,79042,-119596,-86355,0
C00737=40201,41750,-125576,73729,-119771,-89326,0
C00738=40202,41690,-125585,73741,-119796,-89298,0
C00739=36349,45702,-115206,79005,-120009,-86007,0
C00740=41013,41719,-125526,72908,-120217,-89390,0
C00741=40006,41217,-126825,73784,-119389,-89607,0
C00742=35385,45204,-116452,79788,-119187,-86226,0
C00743=36271,45661,-115310,79068,-119941,-86025,0
C00744=35655,46046,-114328,79799,-119764,-85683,0
C00745=36529,46520,-113152,79107,-120530,-85476,0
C00746=42242,41672,-125672,71607,-120788,-89598,0
C00747=39874,40496,-128738,73680,-118845,-90105,0
C00748=34283,45351,-116061,80914,-118604,-85991,0
C00749=35185,45801,-114936,80177,-119362,-85791,0
C00750=34950,46058,-114287,80489,-119342,-85587,0
C00751=35418,46303,-113679,80114,-119744,-85479,0
C00752=35601,46104,-114181,79871,-119759,-85637,0
C00753=36162,45765,-115044,79210,-119929,-85940,0
C00754=36126,45189,-116500,79054,-119616,-86329,0
C00755=40202,41690,-125585,73741,-119796,-89298,0
C00756=40202,41630,-125595,73754,-119821,-89271,0
C00757=36349,45648,-115215,79018,-120028,-85982,0
C00758=41013,41659,-125535,72921,-120243,-89363,0
C00759=40007,41157,-126835,73796,-119416,-89579,0
C00760=35386,45148,-116460,79800,-119207,-86200,0
C00761=36271,45606,-115318,79080,-119960,-86000,0
C00762=35656,45992,-114336,79811,-119782,-85658,0
C00763=36529,46466,-113160,79119,-120549,-85451,0
C00764=42243,41612,-125681,71621,-120815,-89571,0
C00765=39875,40434,-128747,73693,-118872,-90077,0
C00766=34284,45296,-116070,80925,-118623,-85965,0
C00767=35186,45747,-114945,80189,-119379,-85766,0
C00768=34950,46004,-114296,80501,-119359,-85561,0
C00769=35419,46249,-113688,80126,-119763,-85454,0
C00770=35602,46050,-114190,79883,-119778,-85612,0
C00771=36162,45711,-115052,79222,-119948,-85914,0
C00772=36126,45134,-116508,79066,-119635,-86303,0
C00773=40202,41630,-125595,73754,-119821,-89271,0
C00774=40203,41570,-125604,73767,-119848,-89244,0
C00775=36350,45593,-115224,79030,-120048,-85956,0
C00776=41014,41599,-125544,72934,-120269,-89336,0
C00777=40007,41096,-126844,73809,-119441,-89551,0
C00778=35386,45093,-116469,79811,-119225,-86174,0
C00779=36272,45552,-115327,79092,-119980,-85974,0
C00780=35656,45938,-114345,79823,-119801,-85633,0
C00781=36530,46413,-113169,79132,-120567,-85426,0
C00782=42243,41552,-125690,71634,-120843,-89544,0
C00783=39875,40371,-128756,73705,-118899,-90049,0
C00784=34284,45241,-116079,80937,-118641,-85939,0
C00785=35186,45693,-114955,80201,-119397,-85740,0
C00786=34950,45950,-114305,80513,-119378,-85537,0
C00787=35419,46195,-113697,80138,-119781,-85429,0
C00788=35602,45996,-114198,79895,-119796,-85586,0
C00789=36163,45656,-115061,79234,-119967,-85889,0
C00790=36127,45079,-116517,79078,-119655,-86278,0
C00791=40203,41570,-125604,73767,-119848,-89244,0
C00792=40203,41510,-125613,73780,-119873,-89217,0
C00793=36350,45539,-115232,79042,-120066,-85931,0
C00794=41014,41539,-125553,72948,-120296,-89309,0
C00795=40008,41035,-126853,73822,-119467,-89524,0
C00796=35386,45038,-116477,79823,-119244,-86148,0
C00797=36272,45497,-115335,79105,-119999,-85949,0
C00798=35656,45884,-114354,79835,-119819,-85607,0
C00799=36530,46359,-113177,79144,-120587,-85401,0
C00800=42244,41492,-125699,71648,-120870,-89517,0
C00801=39876,40309,-128765,73718,-118925,-90021,0
C00802=34284,45186,-116088,80948,-118658,-85913,0
C00803=35186,45638,-114963,80213,-119416,-85715,0
C00804=34951,45896,-114313,80525,-119395,-85511,0
C00805=35419,46141,-113705,80150,-119798,-85404,0
C00806=35602,45942,-114207,79907,-119814,-85561,0
C00807=36163,45602,-115070,79246,-119987,-85863,0
C00808=36127,45024,-116527,79090,-119674,-86251,0
C00809=40203,41510,-125613,73780,-119873,-89217,0
C00810=40203,41450,-125622,73793,-119898,-89189,0
C00811=36350,45484,-115241,79055,-120086,-85905,0
C00812=41015,41479,-125561,72961,-120322,-89282,0
C00813=40008,40974,-126862,73835,-119494,-89496,0
C00814=35387,44983,-116486,79835,-119263,-86123,0
C00815=36272,45443,-115344,79117,-120018,-85923,0
C00816=35657,45830,-114362,79847,-119837,-85582,0
C00817=36530,46306,-113186,79157,-120605,-85376,0
C00818=42244,41432,-125707,71662,-120898,-89490,0
C00819=39876,40247,-128774,73731,-118951,-89992,0
C00820=34285,45131,-116096,80960,-118677,-85887,0
C00821=35187,45584,-114971,80224,-119434,-85689,0
C00822=34951,45842,-114322,80536,-119413,-85485,0
C00823=35420,46087,-113714,80162,-119817,-85378,0
C00824=35603,45888,-114215,79919,-119833,-85536,0
C00825=36163,45548,-115079,79259,-120005,-85838,0
C00826=36127,44969,-116535,79102,-119694,-86226,0
C00827=40203,41450,-125622,73793,-119898,-89189,0
C00828=40204,41390,-125630,73806,-119925,-89161,0
C00829=36351,45430,-115249,79067,-120105,-85879,0
C00830=41015,41419,-125571,72974,-120349,-89254,0
C00831=40008,40913,-126871,73848,-119519,-89468,0
C00832=35387,44928,-116494,79847,-119281,-86096,0
C00833=36273,45388,-115352,79129,-120037,-85897,0
C00834=35657,45776,-114371,79859,-119857,-85557,0
C00835=36531,46252,-113194,79170,-120623,-85351,0
C00836=42245,41372,-125716,71675,-120924,-89463,0
C00837=39876,40185,-128782,73743,-118978,-89964,0
C00838=34285,45076,-116104,80971,-118694,-85861,0
C00839=35187,45530,-114980,80236,-119452,-85664,0
C00840=34951,45788,-114330,80548,-119432,-85460,0
C00841=35420,46034,-113722,80174,-119835,-85353,0
C00842=35603,45834,-114224,79931,-119851,-85510,0
C00843=36164,45493,-115087,79271,-120025,-85812,0
C00844=36128,44914,-116543,79115,-119713,-86200,0
C00845=40204,41390,-125630,73806,-119925,-89161,0
C00846=40204,41330,-125639,73820,-119950,-89134,0
C00847=36351,45375,-115257,79079,-120125,-85854,0
C00848=41015,41359,-125580,72988,-120375,-89227,0
C00849=40009,40853,-126879,73861,-119546,-89440,0
C00850=35387,44873,-116503,79859,-119301,-86070,0
C00851=36273,45334,-115360,79142,-120057,-85872,0
C00852=35657,45722,-114379,79871,-119875,-85531,0
C00853=36531,46199,-113203,79182,-120643,-85325,0
C00854=42245,41312,-125726,71689,-120952,-89436,0
C00855=39877,40123,-128792,73756,-119004,-89936,0
C00856=34285,45021,-116113,80983,-118712,-85835,0
C00857=35187,45476,-114988,80248,-119471,-85638,0
C00858=34952,45734,-114338,80560,-119449,-85434,0
C00859=35420,45980,-113730,80186,-119853,-85328,0
C00860=35603,45780,-114232,79943,-119870,-85485,0
C00861=36164,45439,-115095,79283,-120043,-85787,0
C00862=36128,44859,-116552,79127,-119733,-86174,0
C00863=40204,41330,-125639,73820,-119950,-89134,0
C00864=40205,41270,-125648,73833,-119975,-89107,0
C00865=36351,45321,-115266,79092,-120143,-85828,0
C00866=41016,41299,-125588,73001,-120402,-89199,0
C00867=40009,40792,-126889,73874,-119571,-89412,0
C00868=35388,44818,-116511,79871,-119319,-86045,0
C00869=36273,45279,-115369,79154,-120075,-85846,0
C00870=35658,45668,-114387,79884,-119894,-85506,0
C00871=36531,46145,-113211,79195,-120661,-85300,0
C00872=42245,41252,-125734,71703,-120980,-89409,0
C00873=39877,40061,-128801,73769,-119032,-89907,0
C00874=34285,44967,-116121,80994,-118731,-85809,0
C00875=35188,45421,-114996,80260,-119489,-85612,0
C00876=34952,45680,-114346,80572,-119467,-85409,0
C00877=35421,45926,-113738,80199,-119872,-85302,0
C00878=35604,45727,-114240,79955,-119888,-85459,0
C00879=36165,45385,-115104,79296,-120063,-85761,0
C00880=36128,44804,-116560,79139,-119751,-86148,0
C00881=40205,41270,-125648,73833,-119975,-89107,0
C00882=40205,41210,-125657,73846,-120002,-89079,0
C00883=36351,45267,-115274,79104,-120163,-85803,0
C00884=41016,41239,-125596,73014,-120428,-89172,0
C00885=40010,40731,-126897,73887,-119597,-89384,0
C00886=35388,44763,-116520,79883,-119339,-86019,0
C00887=36274,45225,-115378,79167,-120095,-85820,0
C00888=35658,45614,-114395,79896,-119912,-85480,0
C00889=36532,46092,-113219,79207,-120680,-85275,0
C00890=42246,41192,-125743,71716,-121007,-89381,0
C00891=39878,39999,-128809,73782,-119058,-89879,0
C00892=34286,44912,-116129,81006,-118748,-85784,0
C00893=35188,45367,-115004,80272,-119508,-85586,0
C00894=34952,45626,-114355,80584,-119486,-85383,0
C00895=35421,45873,-113747,80211,-119889,-85277,0
C00896=35604,45673,-114248,79968,-119907,-85434,0
C00897=36165,45330,-115112,79308,-120082,-85736,0
C00898=36129,44749,-116568,79151,-119771,-86122,0
C00899=40205,41210,-125657,73846,-120002,-89079,0
C00900=40205,41150,-125665,73859,-120027,-89052,0
C00901=36352,45213,-115282,79117,-120182,-85777,0
C00902=41017,41179,-125605,73028,-120454,-89145,0
C00903=40010,40671,-126906,73900,-119624,-89356,0
C00904=35388,44709,-116528,79895,-119357,-85993,0
C00905=36274,45171,-115386,79179,-120114,-85795,0
C00906=35658,45560,-114403,79908,-119930,-85455,0
C00907=36532,46039,-113227,79220,-120699,-85250,0
C00908=42246,41132,-125751,71730,-121035,-89354,0
C00909=39878,39938,-128818,73794,-119085,-89850,0
C00910=34286,44857,-116137,81017,-118766,-85758,0
C00911=35188,45313,-115012,80284,-119526,-85561,0
C00912=34953,45572,-114363,80596,-119503,-85358,0
C00913=35421,45819,-113755,80223,-119907,-85251,0
C00914=35604,45619,-114256,79980,-119926,-85408,0
C00915=36165,45276,-115120,79320,-120101,-85710,0
C00916=36129,44694,-116576,79164,-119790,-86096,0
C00917=40205,41150,-125665,73859,-120027,-89052,0
C00918=40206,41090,-125673,73872,-120053,-89024,0
C00919=36352,45158,-115290,79129,-120202,-85751,0
C00920=41017,41120,-125613,73041,-120480,-89117,0
C00921=40010,40610,-126914,73913,-119649,-89329,0
C00922=35389,44654,-116536,79907,-119377,-85967,0
C00923=36274,45116,-115394,79192,-120134,-85769,0
C00924=35659,45506,-114411,79920,-119949,-85429,0
C00925=36532,45985,-113235,79233,-120718,-85224,0
C00926=42247,41072,-125759,71744,-121062,-89327,0
C00927=39879,39876,-128826,73807,-119111,-89822,0
C00928=34286,44803,-116145,81029,-118785,-85731,0
C00929=35189,45259,-115020,80296,-119544,-85535,0
C00930=34953,45518,-114371,80608,-119521,-85332,0
C00931=35422,45766,-113763,80235,-119926,-85226,0
C00932=35604,45565,-114264,79992,-119944,-85383,0
C00933=36165,45222,-115128,79333,-120120,-85684,0
C00934=36129,44639,-116584,79176,-119810,-86070,0
C00935=40206,41090,-125673,73872,-120053,-89024,0
C00936=40206,41031,-125682,73886,-120079,-88996,0
C00937=36353,45104,-115298,79142,-120220,-85726,0
C00938=41017,41060,-125621,73055,-120506,-89090,0
C00939=40011,40549,-126922,73926,-119675,-89301,0
C00940=35389,44599,-116544,79919,-119395,-85940,0
C00941=36275,45062,-115402,79204,-120152,-85743,0
C00942=35659,45452,-114419,79933,-119967,-85404,0
C00943=36533,45932,-113243,79245,-120737,-85199,0
C00944=42247,41012,-125767,71758,-121090,-89300,0
C00945=39879,39814,-128834,73820,-119139,-89793,0
C00946=34287,44748,-116153,81041,-118802,-85705,0
C00947=35189,45205,-115028,80308,-119563,-85509,0
C00948=34953,45464,-114379,80620,-119540,-85306,0
C00949=35422,45712,-113770,80247,-119944,-85201,0
C00950=35605,45511,-114272,80004,-119963,-85357,0
C00951=36166,45168,-115136,79345,-120138,-85658,0
C00952=36130,44584,-116592,79188,-119829,-86044,0
C00953=40206,41031,-125682,73886,-120079,-88996,0
C00954=40207,40971,-125690,73899,-120104,-88969,0
C00955=36353,45050,-115305,79154,-120240,-85700,0
C00956=41018,41000,-125629,73068,-120533,-89062,0
C00957=40011,40489,-126930,73939,-119702,-89272,0
C00958=35389,44544,-116551,79931,-119414,-85914,0
C00959=36275,45008,-115409,79217,-120172,-85718,0
C00960=35659,45399,-114427,79945,-119986,-85378,0
C00961=36533,45879,-113251,79258,-120756,-85174,0
C00962=42247,40952,-125775,71772,-121118,-89272,0
C00963=39879,39752,-128843,73833,-119165,-89765,0
C00964=34287,44693,-116161,81052,-118820,-85679,0
C00965=35189,45151,-115036,80321,-119581,-85484,0
C00966=34954,45411,-114386,80632,-119557,-85281,0
C00967=35422,45659,-113778,80260,-119963,-85175,0
C00968=35605,45458,-114280,80017,-119981,-85332,0
C00969=36166,45114,-115143,79358,-120158,-85633,0
C00970=36130,44529,-116600,79201,-119849,-86018,0
C00971=40207,40971,-125690,73899,-120104,-88969,0
C00972=40207,40911,-125698,73912,-120130,-88941,0
C00973=36353,44996,-115313,79167,-120259,-85674,0
C00974=41018,40940,-125637,73082,-120559,-89035,0
C00975=40012,40428,-126938,73952,-119727,-89244,0
C00976=35390,44489,-116559,79944,-119433,-85888,0
C00977=36275,44954,-115417,79229,-120191,-85691,0
C00978=35660,45345,-114435,79957,-120005,-85352,0
C00979=36533,45826,-113258,79271,-120774,-85148,0
C00980=42248,40893,-125784,71786,-121145,-89245,0
C00981=39880,39690,-128851,73846,-119192,-89736,0
C00982=34287,44639,-116168,81064,-118839,-85653,0
C00983=35190,45097,-115044,80333,-119600,-85458,0
C00984=34954,45357,-114394,80644,-119575,-85255,0
C00985=35423,45605,-113786,80272,-119981,-85149,0
C00986=35606,45404,-114288,80029,-119999,-85306,0
C00987=36166,45060,-115151,79370,-120178,-85607,0
C00988=36130,44475,-116607,79213,-119868,-85992,0
C00989=40207,40911,-125698,73912,-120130,-88941,0
C00990=40207,40851,-125706,73926,-120156,-88913,0
C00991=36354,44942,-115321,79180,-120279,-85648,0
C00992=41019,40881,-125645,73096,-120585,-89007,0
C00993=40012,40368,-126946,73966,-119754,-89217,0
C00994=35390,44435,-116567,79956,-119452,-85862,0
C00995=36276,44899,-115425,79242,-120211,-85666,0
C00996=35660,45291,-114442,79970,-120024,-85326,0
C00997=36534,45772,-113266,79284,-120793,-85123,0
C00998=42248,40833,-125791,71800,-121172,-89217,0
C00999=39880,39628,-128859,73859,-119218,-89708,0
C01000=34288,44584,-116176,81076,-118856,-85627,0
C01001=35190,45043,-115051,80345,-119618,-85432,0
C01002=34954,45303,-114402,80656,-119594,-85230,0
C01003=35423,45552,-113794,80284,-119999,-85123,0
C01004=35606,45350,-114295,80041,-120018,-85281,0
C01005=36167,45006,-115159,79383,-120196,-85581,0
C01006=36131,44420,-116615,79226,-119888,-85966,0
C01007=40207,40851,-125706,73926,-120156,-88913,0
C01008=40208,40792,-125714,73939,-120182,-88886,0
C01009=36354,44887,-115328,79192,-120298,-85622,0
C01010=41019,40821,-125653,73110,-120612,-88980,0
C01011=40012,40307,-126954,73979,-119780,-89188,0
C01012=35390,44380,-116575,79968,-119471,-85836,0
C01013=36276,44845,-115432,79254,-120230,-85640,0
C01014=35660,45237,-114450,79982,-120042,-85301,0
C01015=36534,45719,-113274,79297,-120812,-85098,0
C01016=42249,40773,-125799,71814,-121199,-89190,0
C01017=39881,39567,-128867,73872,-119246,-89679,0
C01018=34288,44530,-116184,81088,-118874,-85601,0
C01019=35190,44989,-115059,80357,-119636,-85406,0
C01020=34955,45249,-114409,80668,-119611,-85203,0
C01021=35423,45498,-113801,80296,-120017,-85098,0
C01022=35606,45297,-114303,80054,-120036,-85255,0
C01023=36167,44952,-115166,79396,-120215,-85556,0
C01024=36131,44365,-116623,79238,-119907,-85940,0
C01025=40208,40792,-125714,73939,-120182,-88886,0
C01026=40208,40732,-125721,73953,-120207,-88858,0
C01027=36354,44833,-115336,79205,-120317,-85596,0
C01028=41019,40761,-125661,73123,-120639,-88952,0
C01029=40013,40247,-126962,73992,-119806,-89160,0
C01030=35391,44325,-116582,79980,-119490,-85810,0
C01031=36276,44791,-115440,79267,-120249,-85614,0
C01032=35661,45184,-114457,79995,-120060,-85275,0
C01033=36534,45666,-113281,79309,-120831,-85072,0
C01034=42249,40713,-125807,71828,-121227,-89163,0
C01035=39881,39505,-128875,73885,-119272,-89651,0
C01036=34288,44475,-116191,81099,-118893,-85574,0
C01037=35190,44935,-115066,80369,-119655,-85380,0
C01038=34955,45196,-114417,80680,-119629,-85178,0
C01039=35424,45445,-113809,80309,-120035,-85072,0
C01040=35606,45243,-114310,80066,-120055,-85229,0
C01041=36167,44898,-115174,79408,-120235,-85530,0
C01042=36131,44310,-116630,79251,-119927,-85914,0
C01043=40208,40732,-125721,73953,-120207,-88858,0
C01044=40209,40672,-125729,73966,-120234,-88830,0
C01045=36355,44779,-115343,79218,-120336,-85571,0
C01046=41020,40702,-125669,73137,-120666,-88924,0
C01047=40013,40186,-126970,74006,-119832,-89132,0
C01048=35391,44270,-116590,79992,-119509,-85783,0
C01049=36277,44737,-115446,79280,-120268,-85588,0
C01050=35661,45130,-114465,80007,-120079,-85249,0
C01051=36535,45613,-113288,79322,-120850,-85047,0
C01052=42250,40654,-125815,71842,-121254,-89135,0
C01053=39881,39443,-128884,73899,-119298,-89622,0
C01054=34289,44421,-116199,81111,-118910,-85548,0
C01055=35191,44881,-115074,80381,-119673,-85354,0
C01056=34955,45142,-114424,80693,-119648,-85152,0
C01057=35424,45391,-113816,80321,-120053,-85047,0
C01058=35607,45189,-114318,80079,-120073,-85203,0
C01059=36168,44844,-115181,79421,-120253,-85503,0
C01060=36132,44256,-116638,79263,-119947,-85888,0
C01061=40209,40672,-125729,73966,-120234,-88830,0
C01062=40209,40613,-125737,73980,-120259,-88802,0
C01063=36355,44725,-115351,79230,-120356,-85545,0
C01064=41020,40642,-125676,73151,-120692,-88897,0
C01065=40014,40126,-126978,74019,-119858,-89104,0
C01066=35391,44216,-116597,80005,-119528,-85757,0
C01067=36277,44683,-115455,79292,-120288,-85562,0
C01068=35661,45076,-114472,80019,-120097,-85223,0
C01069=36535,45560,-113296,79335,-120869,-85021,0
C01070=42250,40594,-125823,71857,-121282,-89107,0
C01071=39882,39382,-128890,73912,-119326,-89593,0
C01072=34289,44366,-116206,81123,-118928,-85522,0
C01073=35191,44827,-115081,80394,-119691,-85328,0
C01074=34956,45088,-114432,80705,-119666,-85126,0
C01075=35424,45338,-113823,80334,-120072,-85021,0
C01076=35607,45136,-114325,80091,-120091,-85177,0
C01077=36168,44790,-115189,79434,-120273,-85478,0
C01078=36132,44201,-116645,79276,-119966,-85861,0
C01079=40209,40613,-125737,73980,-120259,-88802,0
C01080=40210,40553,-125744,73993,-120286,-88774,0
C01081=36355,44671,-115358,79243,-120375,-85519,0
C01082=41021,40582,-125684,73165,-120719,-88869,0
C01083=40014,40066,-126985,74032,-119885,-89076,0
C01084=35392,44161,-116604,80017,-119547,-85731,0
C01085=36277,44629,-115461,79305,-120307,-85537,0
C01086=35662,45023,-114479,80032,-120117,-85198,0
C01087=36535,45507,-113303,79348,-120888,-84996,0
C01088=42250,40534,-125830,71871,-121309,-89080,0
C01089=39882,39320,-128898,73925,-119352,-89564,0
C01090=34289,44312,-116214,81135,-118947,-85496,0
C01091=35192,44773,-115089,80406,-119710,-85302,0
C01092=34956,45035,-114439,80717,-119683,-85100,0
C01093=35424,45285,-113831,80346,-120090,-84995,0
C01094=35607,45082,-114332,80104,-120111,-85152,0
C01095=36168,44736,-115196,79446,-120292,-85452,0
C01096=36132,44146,-116653,79289,-119986,-85835,0
C01097=40210,40553,-125744,73993,-120286,-88774,0
C01098=40210,40493,-125752,74007,-120311,-88747,0
C01099=36356,44617,-115365,79256,-120395,-85493,0
C01100=41021,40523,-125691,73179,-120745,-88841,0
C01101=40015,40005,-126993,74046,-119911,-89048,0
C01102=35392,44107,-116612,80029,-119566,-85705,0
//INST
///DATE 2025/02/20 16:20
///COMM Generated using RoboDK
///ATTR SC,RW
///GROUP1 RB1
NOP
MOVL C00000 V=30.0 PL=1
MOVL C00001 V=130.0 PL=1
MOVL C00002 V=130.0 PL=1
MOVL C00003 V=30.0 PL=1
MOVL C00004 V=130.0 PL=1
MOVL C00005 V=20.0 PL=1
MOVL C00006 V=130.0 PL=1
MOVL C00007 V=130.0 PL=1
MOVL C00008 V=30.0 PL=1
MOVL C00009 V=130.0 PL=1
MOVL C00010 V=60.0 PL=1
MOVL C00011 V=60.0 PL=1
MOVL C00012 V=60.0 PL=1
MOVL C00013 V=60.0 PL=1
MOVL C00014 V=130.0 PL=1
MOVL C00015 V=30.0 PL=1
MOVL C00016 V=30.0 PL=1
MOVL C00017 V=30.0 PL=1
MOVL C00018 V=30.0 PL=1
MOVL C00019 V=30.0 PL=1
MOVL C00020 V=30.0 PL=1
MOVL C00021 V=30.0 PL=1
MOVL C00022 V=30.0 PL=1
MOVL C00023 V=130.0 PL=1
MOVL C00024 V=130.0 PL=1
MOVL C00025 V=30.0 PL=1
MOVL C00026 V=130.0 PL=1
MOVL C00027 V=20.0 PL=1
MOVL C00028 V=130.0 PL=1
MOVL C00029 V=130.0 PL=1
MOVL C00030 V=30.0 PL=1
MOVL C00031 V=130.0 PL=1
MOVL C00032 V=60.0 PL=1
MOVL C00033 V=60.0 PL=1
MOVL C00034 V=60.0 PL=1
MOVL C00035 V=60.0 PL=1
MOVL C00036 V=130.0 PL=1
MOVL C00037 V=30.0 PL=1
MOVL C00038 V=30.0 PL=1
MOVL C00039 V=30.0 PL=1
MOVL C00040 V=30.0 PL=1
MOVL C00041 V=30.0 PL=1
MOVL C00042 V=30.0 PL=1
MOVL C00043 V=30.0 PL=1
MOVL C00044 V=30.0 PL=1
MOVL C00045 V=130.0 PL=1
MOVL C00046 V=130.0 PL=1
MOVL C00047 V=30.0 PL=1
MOVL C00048 V=130.0 PL=1
MOVL C00049 V=20.0 PL=1
MOVL C00050 V=130.0 PL=1
MOVL C00051 V=130.0 PL=1
MOVL C00052 V=30.0 PL=1
MOVL C00053 V=130.0 PL=1
MOVL C00054 V=60.0 PL=1
MOVL C00055 V=60.0 PL=1
MOVL C00056 V=60.0 PL=1
MOVL C00057 V=60.0 PL=1
MOVL C00058 V=130.0 PL=1
MOVL C00059 V=30.0 PL=1
MOVL C00060 V=30.0 PL=1
MOVL C00061 V=30.0 PL=1
MOVL C00062 V=30.0 PL=1
MOVL C00063 V=30.0 PL=1
MOVL C00064 V=30.0 PL=1
MOVL C00065 V=30.0 PL=1
MOVL C00066 V=30.0 PL=1
MOVL C00067 V=130.0 PL=1
MOVL C00068 V=130.0 PL=1
MOVL C00069 V=30.0 PL=1
MOVL C00070 V=130.0 PL=1
MOVL C00071 V=20.0 PL=1
MOVL C00072 V=130.0 PL=1
MOVL C00073 V=130.0 PL=1
MOVL C00074 V=30.0 PL=1
MOVL C00075 V=130.0 PL=1
MOVL C00076 V=60.0 PL=1
MOVL C00077 V=60.0 PL=1
MOVL C00078 V=60.0 PL=1
MOVL C00079 V=60.0 PL=1
MOVL C00080 V=130.0 PL=1
MOVL C00081 V=30.0 PL=1
MOVL C00082 V=30.0 PL=1
MOVL C00083 V=30.0 PL=1
MOVL C00084 V=30.0 PL=1
MOVL C00085 V=30.0 PL=1
MOVL C00086 V=30.0 PL=1
MOVL C00087 V=30.0 PL=1
MOVL C00088 V=30.0 PL=1
MOVL C00089 V=130.0 PL=1
MOVL C00090 V=130.0 PL=1
MOVL C00091 V=30.0 PL=1
MOVL C00092 V=130.0 PL=1
MOVL C00093 V=20.0 PL=1
MOVL C00094 V=130.0 PL=1
MOVL C00095 V=130.0 PL=1
MOVL C00096 V=30.0 PL=1
MOVL C00097 V=130.0 PL=1
MOVL C00098 V=60.0 PL=1
MOVL C00099 V=60.0 PL=1
MOVL C00100 V=60.0 PL=1
MOVL C00101 V=60.0 PL=1
MOVL C00102 V=130.0 PL=1
MOVL C00103 V=30.0 PL=1
MOVL C00104 V=30.0 PL=1
MOVL C00105 V=30.0 PL=1
MOVL C00106 V=30.0 PL=1
MOVL C00107 V=30.0 PL=1
MOVL C00108 V=30.0 PL=1
MOVL C00109 V=30.0 PL=1
MOVL C00110 V=30.0 PL=1
MOVL C00111 V=130.0 PL=1
MOVL C00112 V=130.0 PL=1
MOVL C00113 V=30.0 PL=1
MOVL C00114 V=130.0 PL=1
MOVL C00115 V=20.0 PL=1
MOVL C00116 V=130.0 PL=1
MOVL C00117 V=130.0 PL=1
MOVL C00118 V=30.0 PL=1
MOVL C00119 V=130.0 PL=1
MOVL C00120 V=60.0 PL=1
MOVL C00121 V=60.0 PL=1
MOVL C00122 V=60.0 PL=1
MOVL C00123 V=60.0 PL=1
MOVL C00124 V=130.0 PL=1
MOVL C00125 V=30.0 PL=1
MOVL C00126 V=30.0 PL=1
MOVL C00127 V=30.0 PL=1
MOVL C00128 V=30.0 PL=1
MOVL C00129 V=30.0 PL=1
MOVL C00130 V=30.0 PL=1
MOVL C00131 V=30.0 PL=1
MOVL C00132 V=30.0 PL=1
MOVL C00133 V=130.0 PL=1
MOVL C00134 V=130.0 PL=1
MOVL C00135 V=30.0 PL=1
MOVL C00136 V=130.0 PL=1
MOVL C00137 V=20.0 PL=1
MOVL C00138 V=130.0 PL=1
MOVL C00139 V=130.0 PL=1
MOVL C00140 V=30.0 PL=1
MOVL C00141 V=130.0 PL=1
MOVL C00142 V=60.0 PL=1
MOVL C00143 V=60.0 PL=1
MOVL C00144 V=60.0 PL=1
MOVL C00145 V=60.0 PL=1
MOVL C00146 V=130.0 PL=1
MOVL C00147 V=30.0 PL=1
MOVL C00148 V=30.0 PL=1
MOVL C00149 V=30.0 PL=1
MOVL C00150 V=30.0 PL=1
MOVL C00151 V=30.0 PL=1
MOVL C00152 V=30.0 PL=1
MOVL C00153 V=30.0 PL=1
MOVL C00154 V=30.0 PL=1
MOVL C00155 V=130.0 PL=1
MOVL C00156 V=130.0 PL=1
MOVL C00157 V=30.0 PL=1
MOVL C00158 V=130.0 PL=1
MOVL C00159 V=20.0 PL=1
MOVL C00160 V=130.0 PL=1
MOVL C00161 V=130.0 PL=1
MOVL C00162 V=30.0 PL=1
MOVL C00163 V=130.0 PL=1
MOVL C00164 V=60.0 PL=1
MOVL C00165 V=60.0 PL=1
MOVL C00166 V=60.0 PL=1
MOVL C00167 V=60.0 PL=1
MOVL C00168 V=130.0 PL=1
MOVL C00169 V=30.0 PL=1
MOVL C00170 V=30.0 PL=1
MOVL C00171 V=30.0 PL=1
MOVL C00172 V=30.0 PL=1
MOVL C00173 V=30.0 PL=1
MOVL C00174 V=30.0 PL=1
MOVL C00175 V=30.0 PL=1
MOVL C00176 V=30.0 PL=1
MOVL C00177 V=130.0 PL=1
MOVL C00178 V=130.0 PL=1
MOVL C00179 V=20.0 PL=1
MOVL C00180 V=130.0 PL=1
MOVL C00181 V=130.0 PL=1
MOVL C00182 V=30.0 PL=1
MOVL C00183 V=130.0 PL=1
MOVL C00184 V=60.0 PL=1
MOVL C00185 V=60.0 PL=1
MOVL C00186 V=60.0 PL=1
MOVL C00187 V=60.0 PL=1
MOVL C00188 V=130.0 PL=1
MOVL C00189 V=30.0 PL=1
MOVL C00190 V=30.0 PL=1
MOVL C00191 V=30.0 PL=1
MOVL C00192 V=30.0 PL=1
MOVL C00193 V=30.0 PL=1
MOVL C00194 V=30.0 PL=1
MOVL C00195 V=30.0 PL=1
MOVL C00196 V=30.0 PL=1
MOVL C00197 V=130.0 PL=1
MOVL C00198 V=130.0 PL=1
MOVL C00199 V=20.0 PL=1
MOVL C00200 V=130.0 PL=1
MOVL C00201 V=130.0 PL=1
MOVL C00202 V=30.0 PL=1
MOVL C00203 V=130.0 PL=1
MOVL C00204 V=60.0 PL=1
MOVL C00205 V=60.0 PL=1
MOVL C00206 V=60.0 PL=1
MOVL C00207 V=60.0 PL=1
MOVL C00208 V=130.0 PL=1
MOVL C00209 V=30.0 PL=1
MOVL C00210 V=30.0 PL=1
MOVL C00211 V=30.0 PL=1
MOVL C00212 V=30.0 PL=1
MOVL C00213 V=30.0 PL=1
MOVL C00214 V=30.0 PL=1
MOVL C00215 V=30.0 PL=1
MOVL C00216 V=30.0 PL=1
MOVL C00217 V=130.0 PL=1
MOVL C00218 V=130.0 PL=1
MOVL C00219 V=20.0 PL=1
MOVL C00220 V=130.0 PL=1
MOVL C00221 V=130.0 PL=1
MOVL C00222 V=30.0 PL=1
MOVL C00223 V=130.0 PL=1
MOVL C00224 V=60.0 PL=1
MOVL C00225 V=60.0 PL=1
MOVL C00226 V=60.0 PL=1
MOVL C00227 V=60.0 PL=1
MOVL C00228 V=130.0 PL=1
MOVL C00229 V=30.0 PL=1
MOVL C00230 V=30.0 PL=1
MOVL C00231 V=30.0 PL=1
MOVL C00232 V=30.0 PL=1
MOVL C00233 V=30.0 PL=1
MOVL C00234 V=30.0 PL=1
MOVL C00235 V=30.0 PL=1
MOVL C00236 V=30.0 PL=1
MOVL C00237 V=130.0 PL=1
MOVL C00238 V=130.0 PL=1
MOVL C00239 V=20.0 PL=1
MOVL C00240 V=130.0 PL=1
MOVL C00241 V=130.0 PL=1
MOVL C00242 V=60.0 PL=1
MOVL C00243 V=60.0 PL=1
MOVL C00244 V=60.0 PL=1
MOVL C00245 V=60.0 PL=1
MOVL C00246 V=130.0 PL=1
MOVL C00247 V=30.0 PL=1
MOVL C00248 V=30.0 PL=1
MOVL C00249 V=30.0 PL=1
MOVL C00250 V=30.0 PL=1
MOVL C00251 V=30.0 PL=1
MOVL C00252 V=30.0 PL=1
MOVL C00253 V=30.0 PL=1
MOVL C00254 V=30.0 PL=1
MOVL C00255 V=130.0 PL=1
MOVL C00256 V=130.0 PL=1
MOVL C00257 V=20.0 PL=1
MOVL C00258 V=130.0 PL=1
MOVL C00259 V=130.0 PL=1
MOVL C00260 V=60.0 PL=1
MOVL C00261 V=60.0 PL=1
MOVL C00262 V=60.0 PL=1
MOVL C00263 V=60.0 PL=1
MOVL C00264 V=130.0 PL=1
MOVL C00265 V=30.0 PL=1
MOVL C00266 V=30.0 PL=1
MOVL C00267 V=30.0 PL=1
MOVL C00268 V=30.0 PL=1
MOVL C00269 V=30.0 PL=1
MOVL C00270 V=30.0 PL=1
MOVL C00271 V=30.0 PL=1
MOVL C00272 V=30.0 PL=1
MOVL C00273 V=130.0 PL=1
MOVL C00274 V=130.0 PL=1
MOVL C00275 V=20.0 PL=1
MOVL C00276 V=130.0 PL=1
MOVL C00277 V=130.0 PL=1
MOVL C00278 V=60.0 PL=1
MOVL C00279 V=60.0 PL=1
MOVL C00280 V=60.0 PL=1
MOVL C00281 V=60.0 PL=1
MOVL C00282 V=130.0 PL=1
MOVL C00283 V=30.0 PL=1
MOVL C00284 V=30.0 PL=1
MOVL C00285 V=30.0 PL=1
MOVL C00286 V=30.0 PL=1
MOVL C00287 V=30.0 PL=1
MOVL C00288 V=30.0 PL=1
MOVL C00289 V=30.0 PL=1
MOVL C00290 V=30.0 PL=1
MOVL C00291 V=130.0 PL=1
MOVL C00292 V=130.0 PL=1
MOVL C00293 V=20.0 PL=1
MOVL C00294 V=130.0 PL=1
MOVL C00295 V=130.0 PL=1
MOVL C00296 V=60.0 PL=1
MOVL C00297 V=60.0 PL=1
MOVL C00298 V=60.0 PL=1
MOVL C00299 V=60.0 PL=1
MOVL C00300 V=130.0 PL=1
MOVL C00301 V=30.0 PL=1
MOVL C00302 V=30.0 PL=1
MOVL C00303 V=30.0 PL=1
MOVL C00304 V=30.0 PL=1
MOVL C00305 V=30.0 PL=1
MOVL C00306 V=30.0 PL=1
MOVL C00307 V=30.0 PL=1
MOVL C00308 V=30.0 PL=1
MOVL C00309 V=130.0 PL=1
MOVL C00310 V=130.0 PL=1
MOVL C00311 V=20.0 PL=1
MOVL C00312 V=130.0 PL=1
MOVL C00313 V=130.0 PL=1
MOVL C00314 V=60.0 PL=1
MOVL C00315 V=60.0 PL=1
MOVL C00316 V=60.0 PL=1
MOVL C00317 V=60.0 PL=1
MOVL C00318 V=130.0 PL=1
MOVL C00319 V=30.0 PL=1
MOVL C00320 V=30.0 PL=1
MOVL C00321 V=30.0 PL=1
MOVL C00322 V=30.0 PL=1
MOVL C00323 V=30.0 PL=1
MOVL C00324 V=30.0 PL=1
MOVL C00325 V=30.0 PL=1
MOVL C00326 V=30.0 PL=1
MOVL C00327 V=130.0 PL=1
MOVL C00328 V=130.0 PL=1
MOVL C00329 V=20.0 PL=1
MOVL C00330 V=130.0 PL=1
MOVL C00331 V=130.0 PL=1
MOVL C00332 V=60.0 PL=1
MOVL C00333 V=60.0 PL=1
MOVL C00334 V=60.0 PL=1
MOVL C00335 V=60.0 PL=1
MOVL C00336 V=130.0 PL=1
MOVL C00337 V=30.0 PL=1
MOVL C00338 V=30.0 PL=1
MOVL C00339 V=30.0 PL=1
MOVL C00340 V=30.0 PL=1
MOVL C00341 V=30.0 PL=1
MOVL C00342 V=30.0 PL=1
MOVL C00343 V=30.0 PL=1
MOVL C00344 V=30.0 PL=1
MOVL C00345 V=130.0 PL=1
MOVL C00346 V=130.0 PL=1
MOVL C00347 V=20.0 PL=1
MOVL C00348 V=130.0 PL=1
MOVL C00349 V=130.0 PL=1
MOVL C00350 V=60.0 PL=1
MOVL C00351 V=60.0 PL=1
MOVL C00352 V=60.0 PL=1
MOVL C00353 V=60.0 PL=1
MOVL C00354 V=130.0 PL=1
MOVL C00355 V=30.0 PL=1
MOVL C00356 V=30.0 PL=1
MOVL C00357 V=30.0 PL=1
MOVL C00358 V=30.0 PL=1
MOVL C00359 V=30.0 PL=1
MOVL C00360 V=30.0 PL=1
MOVL C00361 V=30.0 PL=1
MOVL C00362 V=30.0 PL=1
MOVL C00363 V=130.0 PL=1
MOVL C00364 V=130.0 PL=1
MOVL C00365 V=20.0 PL=1
MOVL C00366 V=130.0 PL=1
MOVL C00367 V=130.0 PL=1
MOVL C00368 V=60.0 PL=1
MOVL C00369 V=60.0 PL=1
MOVL C00370 V=60.0 PL=1
MOVL C00371 V=60.0 PL=1
MOVL C00372 V=130.0 PL=1
MOVL C00373 V=30.0 PL=1
MOVL C00374 V=30.0 PL=1
MOVL C00375 V=30.0 PL=1
MOVL C00376 V=30.0 PL=1
MOVL C00377 V=30.0 PL=1
MOVL C00378 V=30.0 PL=1
MOVL C00379 V=30.0 PL=1
MOVL C00380 V=30.0 PL=1
MOVL C00381 V=130.0 PL=1
MOVL C00382 V=130.0 PL=1
MOVL C00383 V=20.0 PL=1
MOVL C00384 V=130.0 PL=1
MOVL C00385 V=130.0 PL=1
MOVL C00386 V=60.0 PL=1
MOVL C00387 V=60.0 PL=1
MOVL C00388 V=60.0 PL=1
MOVL C00389 V=60.0 PL=1
MOVL C00390 V=130.0 PL=1
MOVL C00391 V=30.0 PL=1
MOVL C00392 V=30.0 PL=1
MOVL C00393 V=30.0 PL=1
MOVL C00394 V=30.0 PL=1
MOVL C00395 V=30.0 PL=1
MOVL C00396 V=30.0 PL=1
MOVL C00397 V=30.0 PL=1
MOVL C00398 V=30.0 PL=1
MOVL C00399 V=130.0 PL=1
MOVL C00400 V=130.0 PL=1
MOVL C00401 V=30.0 PL=1
MOVL C00402 V=130.0 PL=1
MOVL C00403 V=30.0 PL=1
MOVL C00404 V=130.0 PL=1
MOVL C00405 V=20.0 PL=1
MOVL C00406 V=130.0 PL=1
MOVL C00407 V=130.0 PL=1
MOVL C00408 V=60.0 PL=1
MOVL C00409 V=60.0 PL=1
MOVL C00410 V=60.0 PL=1
MOVL C00411 V=60.0 PL=1
MOVL C00412 V=130.0 PL=1
MOVL C00413 V=30.0 PL=1
MOVL C00414 V=30.0 PL=1
MOVL C00415 V=30.0 PL=1
MOVL C00416 V=30.0 PL=1
MOVL C00417 V=30.0 PL=1
MOVL C00418 V=30.0 PL=1
MOVL C00419 V=30.0 PL=1
MOVL C00420 V=30.0 PL=1
MOVL C00421 V=130.0 PL=1
MOVL C00422 V=130.0 PL=1
MOVL C00423 V=30.0 PL=1
MOVL C00424 V=130.0 PL=1
MOVL C00425 V=30.0 PL=1
MOVL C00426 V=130.0 PL=1
MOVL C00427 V=20.0 PL=1
MOVL C00428 V=130.0 PL=1
MOVL C00429 V=130.0 PL=1
MOVL C00430 V=60.0 PL=1
MOVL C00431 V=60.0 PL=1
MOVL C00432 V=60.0 PL=1
MOVL C00433 V=60.0 PL=1
MOVL C00434 V=130.0 PL=1
MOVL C00435 V=30.0 PL=1
MOVL C00436 V=30.0 PL=1
MOVL C00437 V=30.0 PL=1
MOVL C00438 V=30.0 PL=1
MOVL C00439 V=30.0 PL=1
MOVL C00440 V=30.0 PL=1
MOVL C00441 V=30.0 PL=1
MOVL C00442 V=30.0 PL=1
MOVL C00443 V=130.0 PL=1
MOVL C00444 V=130.0 PL=1
MOVL C00445 V=20.0 PL=1
MOVL C00446 V=130.0 PL=1
MOVL C00447 V=130.0 PL=1
MOVL C00448 V=60.0 PL=1
MOVL C00449 V=60.0 PL=1
MOVL C00450 V=60.0 PL=1
MOVL C00451 V=60.0 PL=1
MOVL C00452 V=130.0 PL=1
MOVL C00453 V=30.0 PL=1
MOVL C00454 V=30.0 PL=1
MOVL C00455 V=30.0 PL=1
MOVL C00456 V=30.0 PL=1
MOVL C00457 V=30.0 PL=1
MOVL C00458 V=30.0 PL=1
MOVL C00459 V=30.0 PL=1
MOVL C00460 V=30.0 PL=1
MOVL C00461 V=130.0 PL=1
MOVL C00462 V=130.0 PL=1
MOVL C00463 V=20.0 PL=1
MOVL C00464 V=130.0 PL=1
MOVL C00465 V=130.0 PL=1
MOVL C00466 V=60.0 PL=1
MOVL C00467 V=60.0 PL=1
MOVL C00468 V=60.0 PL=1
MOVL C00469 V=60.0 PL=1
MOVL C00470 V=130.0 PL=1
MOVL C00471 V=30.0 PL=1
MOVL C00472 V=30.0 PL=1
MOVL C00473 V=30.0 PL=1
MOVL C00474 V=30.0 PL=1
MOVL C00475 V=30.0 PL=1
MOVL C00476 V=30.0 PL=1
MOVL C00477 V=30.0 PL=1
MOVL C00478 V=30.0 PL=1
MOVL C00479 V=130.0 PL=1
MOVL C00480 V=130.0 PL=1
MOVL C00481 V=20.0 PL=1
MOVL C00482 V=130.0 PL=1
MOVL C00483 V=130.0 PL=1
MOVL C00484 V=60.0 PL=1
MOVL C00485 V=60.0 PL=1
MOVL C00486 V=60.0 PL=1
MOVL C00487 V=60.0 PL=1
MOVL C00488 V=130.0 PL=1
MOVL C00489 V=30.0 PL=1
MOVL C00490 V=30.0 PL=1
MOVL C00491 V=30.0 PL=1
MOVL C00492 V=30.0 PL=1
MOVL C00493 V=30.0 PL=1
MOVL C00494 V=30.0 PL=1
MOVL C00495 V=30.0 PL=1
MOVL C00496 V=30.0 PL=1
MOVL C00497 V=130.0 PL=1
MOVL C00498 V=130.0 PL=1
MOVL C00499 V=20.0 PL=1
MOVL C00500 V=130.0 PL=1
MOVL C00501 V=130.0 PL=1
MOVL C00502 V=60.0 PL=1
MOVL C00503 V=60.0 PL=1
MOVL C00504 V=60.0 PL=1
MOVL C00505 V=60.0 PL=1
MOVL C00506 V=130.0 PL=1
MOVL C00507 V=30.0 PL=1
MOVL C00508 V=30.0 PL=1
MOVL C00509 V=30.0 PL=1
MOVL C00510 V=30.0 PL=1
MOVL C00511 V=30.0 PL=1
MOVL C00512 V=30.0 PL=1
MOVL C00513 V=30.0 PL=1
MOVL C00514 V=30.0 PL=1
MOVL C00515 V=130.0 PL=1
MOVL C00516 V=130.0 PL=1
MOVL C00517 V=30.0 PL=1
MOVL C00518 V=130.0 PL=1
MOVL C00519 V=20.0 PL=1
MOVL C00520 V=130.0 PL=1
MOVL C00521 V=130.0 PL=1
MOVL C00522 V=60.0 PL=1
MOVL C00523 V=60.0 PL=1
MOVL C00524 V=60.0 PL=1
MOVL C00525 V=60.0 PL=1
MOVL C00526 V=130.0 PL=1
MOVL C00527 V=30.0 PL=1
MOVL C00528 V=30.0 PL=1
MOVL C00529 V=30.0 PL=1
MOVL C00530 V=30.0 PL=1
MOVL C00531 V=30.0 PL=1
MOVL C00532 V=30.0 PL=1
MOVL C00533 V=30.0 PL=1
MOVL C00534 V=30.0 PL=1
MOVL C00535 V=130.0 PL=1
MOVL C00536 V=130.0 PL=1
MOVL C00537 V=20.0 PL=1
MOVL C00538 V=130.0 PL=1
MOVL C00539 V=130.0 PL=1
MOVL C00540 V=60.0 PL=1
MOVL C00541 V=60.0 PL=1
MOVL C00542 V=60.0 PL=1
MOVL C00543 V=60.0 PL=1
MOVL C00544 V=130.0 PL=1
MOVL C00545 V=30.0 PL=1
MOVL C00546 V=30.0 PL=1
MOVL C00547 V=30.0 PL=1
MOVL C00548 V=30.0 PL=1
MOVL C00549 V=30.0 PL=1
MOVL C00550 V=30.0 PL=1
MOVL C00551 V=30.0 PL=1
MOVL C00552 V=30.0 PL=1
MOVL C00553 V=130.0 PL=1
MOVL C00554 V=130.0 PL=1
MOVL C00555 V=20.0 PL=1
MOVL C00556 V=130.0 PL=1
MOVL C00557 V=130.0 PL=1
MOVL C00558 V=60.0 PL=1
MOVL C00559 V=60.0 PL=1
MOVL C00560 V=60.0 PL=1
MOVL C00561 V=60.0 PL=1
MOVL C00562 V=130.0 PL=1
MOVL C00563 V=30.0 PL=1
MOVL C00564 V=30.0 PL=1
MOVL C00565 V=30.0 PL=1
MOVL C00566 V=30.0 PL=1
MOVL C00567 V=30.0 PL=1
MOVL C00568 V=30.0 PL=1
MOVL C00569 V=30.0 PL=1
MOVL C00570 V=30.0 PL=1
MOVL C00571 V=130.0 PL=1
MOVL C00572 V=130.0 PL=1
MOVL C00573 V=20.0 PL=1
MOVL C00574 V=130.0 PL=1
MOVL C00575 V=130.0 PL=1
MOVL C00576 V=30.0 PL=1
MOVL C00577 V=130.0 PL=1
MOVL C00578 V=60.0 PL=1
MOVL C00579 V=60.0 PL=1
MOVL C00580 V=60.0 PL=1
MOVL C00581 V=60.0 PL=1
MOVL C00582 V=130.0 PL=1
MOVL C00583 V=30.0 PL=1
MOVL C00584 V=30.0 PL=1
MOVL C00585 V=30.0 PL=1
MOVL C00586 V=30.0 PL=1
MOVL C00587 V=30.0 PL=1
MOVL C00588 V=30.0 PL=1
MOVL C00589 V=30.0 PL=1
MOVL C00590 V=30.0 PL=1
MOVL C00591 V=130.0 PL=1
MOVL C00592 V=130.0 PL=1
MOVL C00593 V=20.0 PL=1
MOVL C00594 V=130.0 PL=1
MOVL C00595 V=130.0 PL=1
MOVL C00596 V=60.0 PL=1
MOVL C00597 V=60.0 PL=1
MOVL C00598 V=60.0 PL=1
MOVL C00599 V=60.0 PL=1
MOVL C00600 V=130.0 PL=1
MOVL C00601 V=30.0 PL=1
MOVL C00602 V=30.0 PL=1
MOVL C00603 V=30.0 PL=1
MOVL C00604 V=30.0 PL=1
MOVL C00605 V=30.0 PL=1
MOVL C00606 V=30.0 PL=1
MOVL C00607 V=30.0 PL=1
MOVL C00608 V=30.0 PL=1
MOVL C00609 V=130.0 PL=1
MOVL C00610 V=130.0 PL=1
MOVL C00611 V=20.0 PL=1
MOVL C00612 V=130.0 PL=1
MOVL C00613 V=130.0 PL=1
MOVL C00614 V=60.0 PL=1
MOVL C00615 V=60.0 PL=1
MOVL C00616 V=60.0 PL=1
MOVL C00617 V=60.0 PL=1
MOVL C00618 V=130.0 PL=1
MOVL C00619 V=30.0 PL=1
MOVL C00620 V=30.0 PL=1
MOVL C00621 V=30.0 PL=1
MOVL C00622 V=30.0 PL=1
MOVL C00623 V=30.0 PL=1
MOVL C00624 V=30.0 PL=1
MOVL C00625 V=30.0 PL=1
MOVL C00626 V=30.0 PL=1
MOVL C00627 V=130.0 PL=1
MOVL C00628 V=130.0 PL=1
MOVL C00629 V=20.0 PL=1
MOVL C00630 V=130.0 PL=1
MOVL C00631 V=130.0 PL=1
MOVL C00632 V=60.0 PL=1
MOVL C00633 V=60.0 PL=1
MOVL C00634 V=60.0 PL=1
MOVL C00635 V=60.0 PL=1
MOVL C00636 V=130.0 PL=1
MOVL C00637 V=30.0 PL=1
MOVL C00638 V=30.0 PL=1
MOVL C00639 V=30.0 PL=1
MOVL C00640 V=30.0 PL=1
MOVL C00641 V=30.0 PL=1
MOVL C00642 V=30.0 PL=1
MOVL C00643 V=30.0 PL=1
MOVL C00644 V=30.0 PL=1
MOVL C00645 V=130.0 PL=1
MOVL C00646 V=130.0 PL=1
MOVL C00647 V=20.0 PL=1
MOVL C00648 V=130.0 PL=1
MOVL C00649 V=130.0 PL=1
MOVL C00650 V=60.0 PL=1
MOVL C00651 V=60.0 PL=1
MOVL C00652 V=60.0 PL=1
MOVL C00653 V=60.0 PL=1
MOVL C00654 V=130.0 PL=1
MOVL C00655 V=30.0 PL=1
MOVL C00656 V=30.0 PL=1
MOVL C00657 V=30.0 PL=1
MOVL C00658 V=30.0 PL=1
MOVL C00659 V=30.0 PL=1
MOVL C00660 V=30.0 PL=1
MOVL C00661 V=30.0 PL=1
MOVL C00662 V=30.0 PL=1
MOVL C00663 V=130.0 PL=1
MOVL C00664 V=130.0 PL=1
MOVL C00665 V=20.0 PL=1
MOVL C00666 V=130.0 PL=1
MOVL C00667 V=130.0 PL=1
MOVL C00668 V=60.0 PL=1
MOVL C00669 V=60.0 PL=1
MOVL C00670 V=60.0 PL=1
MOVL C00671 V=60.0 PL=1
MOVL C00672 V=130.0 PL=1
MOVL C00673 V=30.0 PL=1
MOVL C00674 V=30.0 PL=1
MOVL C00675 V=30.0 PL=1
MOVL C00676 V=30.0 PL=1
MOVL C00677 V=30.0 PL=1
MOVL C00678 V=30.0 PL=1
MOVL C00679 V=30.0 PL=1
MOVL C00680 V=30.0 PL=1
MOVL C00681 V=130.0 PL=1
MOVL C00682 V=130.0 PL=1
MOVL C00683 V=20.0 PL=1
MOVL C00684 V=130.0 PL=1
MOVL C00685 V=130.0 PL=1
MOVL C00686 V=60.0 PL=1
MOVL C00687 V=60.0 PL=1
MOVL C00688 V=60.0 PL=1
MOVL C00689 V=60.0 PL=1
MOVL C00690 V=130.0 PL=1
MOVL C00691 V=30.0 PL=1
MOVL C00692 V=30.0 PL=1
MOVL C00693 V=30.0 PL=1
MOVL C00694 V=30.0 PL=1
MOVL C00695 V=30.0 PL=1
MOVL C00696 V=30.0 PL=1
MOVL C00697 V=30.0 PL=1
MOVL C00698 V=30.0 PL=1
MOVL C00699 V=130.0 PL=1
MOVL C00700 V=130.0 PL=1
MOVL C00701 V=20.0 PL=1
MOVL C00702 V=130.0 PL=1
MOVL C00703 V=130.0 PL=1
MOVL C00704 V=60.0 PL=1
MOVL C00705 V=60.0 PL=1
MOVL C00706 V=60.0 PL=1
MOVL C00707 V=60.0 PL=1
MOVL C00708 V=130.0 PL=1
MOVL C00709 V=30.0 PL=1
MOVL C00710 V=30.0 PL=1
MOVL C00711 V=30.0 PL=1
MOVL C00712 V=30.0 PL=1
MOVL C00713 V=30.0 PL=1
MOVL C00714 V=30.0 PL=1
MOVL C00715 V=30.0 PL=1
MOVL C00716 V=30.0 PL=1
MOVL C00717 V=130.0 PL=1
MOVL C00718 V=130.0 PL=1
MOVL C00719 V=20.0 PL=1
MOVL C00720 V=130.0 PL=1
MOVL C00721 V=130.0 PL=1
MOVL C00722 V=60.0 PL=1
MOVL C00723 V=60.0 PL=1
MOVL C00724 V=60.0 PL=1
MOVL C00725 V=60.0 PL=1
MOVL C00726 V=130.0 PL=1
MOVL C00727 V=30.0 PL=1
MOVL C00728 V=30.0 PL=1
MOVL C00729 V=30.0 PL=1
MOVL C00730 V=30.0 PL=1
MOVL C00731 V=30.0 PL=1
MOVL C00732 V=30.0 PL=1
MOVL C00733 V=30.0 PL=1
MOVL C00734 V=30.0 PL=1
MOVL C00735 V=130.0 PL=1
MOVL C00736 V=130.0 PL=1
MOVL C00737 V=20.0 PL=1
MOVL C00738 V=130.0 PL=1
MOVL C00739 V=130.0 PL=1
MOVL C00740 V=60.0 PL=1
MOVL C00741 V=60.0 PL=1
MOVL C00742 V=60.0 PL=1
MOVL C00743 V=60.0 PL=1
MOVL C00744 V=130.0 PL=1
MOVL C00745 V=30.0 PL=1
MOVL C00746 V=30.0 PL=1
MOVL C00747 V=30.0 PL=1
MOVL C00748 V=30.0 PL=1
MOVL C00749 V=30.0 PL=1
MOVL C00750 V=30.0 PL=1
MOVL C00751 V=30.0 PL=1
MOVL C00752 V=30.0 PL=1
MOVL C00753 V=130.0 PL=1
MOVL C00754 V=130.0 PL=1
MOVL C00755 V=20.0 PL=1
MOVL C00756 V=130.0 PL=1
MOVL C00757 V=130.0 PL=1
MOVL C00758 V=60.0 PL=1
MOVL C00759 V=60.0 PL=1
MOVL C00760 V=60.0 PL=1
MOVL C00761 V=60.0 PL=1
MOVL C00762 V=130.0 PL=1
MOVL C00763 V=30.0 PL=1
MOVL C00764 V=30.0 PL=1
MOVL C00765 V=30.0 PL=1
MOVL C00766 V=30.0 PL=1
MOVL C00767 V=30.0 PL=1
MOVL C00768 V=30.0 PL=1
MOVL C00769 V=30.0 PL=1
MOVL C00770 V=30.0 PL=1
MOVL C00771 V=130.0 PL=1
MOVL C00772 V=130.0 PL=1
MOVL C00773 V=20.0 PL=1
MOVL C00774 V=130.0 PL=1
MOVL C00775 V=130.0 PL=1
MOVL C00776 V=60.0 PL=1
MOVL C00777 V=60.0 PL=1
MOVL C00778 V=60.0 PL=1
MOVL C00779 V=60.0 PL=1
MOVL C00780 V=130.0 PL=1
MOVL C00781 V=30.0 PL=1
MOVL C00782 V=30.0 PL=1
MOVL C00783 V=30.0 PL=1
MOVL C00784 V=30.0 PL=1
MOVL C00785 V=30.0 PL=1
MOVL C00786 V=30.0 PL=1
MOVL C00787 V=30.0 PL=1
MOVL C00788 V=30.0 PL=1
MOVL C00789 V=130.0 PL=1
MOVL C00790 V=130.0 PL=1
MOVL C00791 V=20.0 PL=1
MOVL C00792 V=130.0 PL=1
MOVL C00793 V=130.0 PL=1
MOVL C00794 V=60.0 PL=1
MOVL C00795 V=60.0 PL=1
MOVL C00796 V=60.0 PL=1
MOVL C00797 V=60.0 PL=1
MOVL C00798 V=130.0 PL=1
MOVL C00799 V=30.0 PL=1
MOVL C00800 V=30.0 PL=1
MOVL C00801 V=30.0 PL=1
MOVL C00802 V=30.0 PL=1
MOVL C00803 V=30.0 PL=1
MOVL C00804 V=30.0 PL=1
MOVL C00805 V=30.0 PL=1
MOVL C00806 V=30.0 PL=1
MOVL C00807 V=130.0 PL=1
MOVL C00808 V=130.0 PL=1
MOVL C00809 V=20.0 PL=1
MOVL C00810 V=130.0 PL=1
MOVL C00811 V=130.0 PL=1
MOVL C00812 V=60.0 PL=1
MOVL C00813 V=60.0 PL=1
MOVL C00814 V=60.0 PL=1
MOVL C00815 V=60.0 PL=1
MOVL C00816 V=130.0 PL=1
MOVL C00817 V=30.0 PL=1
MOVL C00818 V=30.0 PL=1
MOVL C00819 V=30.0 PL=1
MOVL C00820 V=30.0 PL=1
MOVL C00821 V=30.0 PL=1
MOVL C00822 V=30.0 PL=1
MOVL C00823 V=30.0 PL=1
MOVL C00824 V=30.0 PL=1
MOVL C00825 V=130.0 PL=1
MOVL C00826 V=130.0 PL=1
MOVL C00827 V=20.0 PL=1
MOVL C00828 V=130.0 PL=1
MOVL C00829 V=130.0 PL=1
MOVL C00830 V=60.0 PL=1
MOVL C00831 V=60.0 PL=1
MOVL C00832 V=60.0 PL=1
MOVL C00833 V=60.0 PL=1
MOVL C00834 V=130.0 PL=1
MOVL C00835 V=30.0 PL=1
MOVL C00836 V=30.0 PL=1
MOVL C00837 V=30.0 PL=1
MOVL C00838 V=30.0 PL=1
MOVL C00839 V=30.0 PL=1
MOVL C00840 V=30.0 PL=1
MOVL C00841 V=30.0 PL=1
MOVL C00842 V=30.0 PL=1
MOVL C00843 V=130.0 PL=1
MOVL C00844 V=130.0 PL=1
MOVL C00845 V=20.0 PL=1
MOVL C00846 V=130.0 PL=1
MOVL C00847 V=130.0 PL=1
MOVL C00848 V=60.0 PL=1
MOVL C00849 V=60.0 PL=1
MOVL C00850 V=60.0 PL=1
MOVL C00851 V=60.0 PL=1
MOVL C00852 V=130.0 PL=1
MOVL C00853 V=30.0 PL=1
MOVL C00854 V=30.0 PL=1
MOVL C00855 V=30.0 PL=1
MOVL C00856 V=30.0 PL=1
MOVL C00857 V=30.0 PL=1
MOVL C00858 V=30.0 PL=1
MOVL C00859 V=30.0 PL=1
MOVL C00860 V=30.0 PL=1
MOVL C00861 V=130.0 PL=1
MOVL C00862 V=130.0 PL=1
MOVL C00863 V=20.0 PL=1
MOVL C00864 V=130.0 PL=1
MOVL C00865 V=130.0 PL=1
MOVL C00866 V=60.0 PL=1
MOVL C00867 V=60.0 PL=1
MOVL C00868 V=60.0 PL=1
MOVL C00869 V=60.0 PL=1
MOVL C00870 V=130.0 PL=1
MOVL C00871 V=30.0 PL=1
MOVL C00872 V=30.0 PL=1
MOVL C00873 V=30.0 PL=1
MOVL C00874 V=30.0 PL=1
MOVL C00875 V=30.0 PL=1
MOVL C00876 V=30.0 PL=1
MOVL C00877 V=30.0 PL=1
MOVL C00878 V=30.0 PL=1
MOVL C00879 V=130.0 PL=1
MOVL C00880 V=130.0 PL=1
MOVL C00881 V=20.0 PL=1
MOVL C00882 V=130.0 PL=1
MOVL C00883 V=130.0 PL=1
MOVL C00884 V=60.0 PL=1
MOVL C00885 V=60.0 PL=1
MOVL C00886 V=60.0 PL=1
MOVL C00887 V=60.0 PL=1
MOVL C00888 V=130.0 PL=1
MOVL C00889 V=30.0 PL=1
MOVL C00890 V=30.0 PL=1
MOVL C00891 V=30.0 PL=1
MOVL C00892 V=30.0 PL=1
MOVL C00893 V=30.0 PL=1
MOVL C00894 V=30.0 PL=1
MOVL C00895 V=30.0 PL=1
MOVL C00896 V=30.0 PL=1
MOVL C00897 V=130.0 PL=1
MOVL C00898 V=130.0 PL=1
MOVL C00899 V=20.0 PL=1
MOVL C00900 V=130.0 PL=1
MOVL C00901 V=130.0 PL=1
MOVL C00902 V=60.0 PL=1
MOVL C00903 V=60.0 PL=1
MOVL C00904 V=60.0 PL=1
MOVL C00905 V=60.0 PL=1
MOVL C00906 V=130.0 PL=1
MOVL C00907 V=30.0 PL=1
MOVL C00908 V=30.0 PL=1
MOVL C00909 V=30.0 PL=1
MOVL C00910 V=30.0 PL=1
MOVL C00911 V=30.0 PL=1
MOVL C00912 V=30.0 PL=1
MOVL C00913 V=30.0 PL=1
MOVL C00914 V=30.0 PL=1
MOVL C00915 V=130.0 PL=1
MOVL C00916 V=130.0 PL=1
MOVL C00917 V=20.0 PL=1
MOVL C00918 V=130.0 PL=1
MOVL C00919 V=130.0 PL=1
MOVL C00920 V=60.0 PL=1
MOVL C00921 V=60.0 PL=1
MOVL C00922 V=60.0 PL=1
MOVL C00923 V=60.0 PL=1
MOVL C00924 V=130.0 PL=1
MOVL C00925 V=30.0 PL=1
MOVL C00926 V=30.0 PL=1
MOVL C00927 V=30.0 PL=1
MOVL C00928 V=30.0 PL=1
MOVL C00929 V=30.0 PL=1
MOVL C00930 V=30.0 PL=1
MOVL C00931 V=30.0 PL=1
MOVL C00932 V=30.0 PL=1
MOVL C00933 V=130.0 PL=1
MOVL C00934 V=130.0 PL=1
MOVL C00935 V=20.0 PL=1
MOVL C00936 V=130.0 PL=1
MOVL C00937 V=130.0 PL=1
MOVL C00938 V=60.0 PL=1
MOVL C00939 V=60.0 PL=1
MOVL C00940 V=60.0 PL=1
MOVL C00941 V=60.0 PL=1
MOVL C00942 V=130.0 PL=1
MOVL C00943 V=30.0 PL=1
MOVL C00944 V=30.0 PL=1
MOVL C00945 V=30.0 PL=1
MOVL C00946 V=30.0 PL=1
MOVL C00947 V=30.0 PL=1
MOVL C00948 V=30.0 PL=1
MOVL C00949 V=30.0 PL=1
MOVL C00950 V=30.0 PL=1
MOVL C00951 V=130.0 PL=1
MOVL C00952 V=130.0 PL=1
MOVL C00953 V=20.0 PL=1
MOVL C00954 V=130.0 PL=1
MOVL C00955 V=130.0 PL=1
MOVL C00956 V=60.0 PL=1
MOVL C00957 V=60.0 PL=1
MOVL C00958 V=60.0 PL=1
MOVL C00959 V=60.0 PL=1
MOVL C00960 V=130.0 PL=1
MOVL C00961 V=30.0 PL=1
MOVL C00962 V=30.0 PL=1
MOVL C00963 V=30.0 PL=1
MOVL C00964 V=30.0 PL=1
MOVL C00965 V=30.0 PL=1
MOVL C00966 V=30.0 PL=1
MOVL C00967 V=30.0 PL=1
MOVL C00968 V=30.0 PL=1
MOVL C00969 V=130.0 PL=1
MOVL C00970 V=130.0 PL=1
MOVL C00971 V=20.0 PL=1
MOVL C00972 V=130.0 PL=1
MOVL C00973 V=130.0 PL=1
MOVL C00974 V=60.0 PL=1
MOVL C00975 V=60.0 PL=1
MOVL C00976 V=60.0 PL=1
MOVL C00977 V=60.0 PL=1
MOVL C00978 V=130.0 PL=1
MOVL C00979 V=30.0 PL=1
MOVL C00980 V=30.0 PL=1
MOVL C00981 V=30.0 PL=1
MOVL C00982 V=30.0 PL=1
MOVL C00983 V=30.0 PL=1
MOVL C00984 V=30.0 PL=1
MOVL C00985 V=30.0 PL=1
MOVL C00986 V=30.0 PL=1
MOVL C00987 V=130.0 PL=1
MOVL C00988 V=130.0 PL=1
MOVL C00989 V=20.0 PL=1
MOVL C00990 V=130.0 PL=1
MOVL C00991 V=130.0 PL=1
MOVL C00992 V=60.0 PL=1
MOVL C00993 V=60.0 PL=1
MOVL C00994 V=60.0 PL=1
MOVL C00995 V=60.0 PL=1
MOVL C00996 V=130.0 PL=1
MOVL C00997 V=30.0 PL=1
MOVL C00998 V=30.0 PL=1
MOVL C00999 V=30.0 PL=1
MOVL C01000 V=30.0 PL=1
MOVL C01001 V=30.0 PL=1
MOVL C01002 V=30.0 PL=1
MOVL C01003 V=30.0 PL=1
MOVL C01004 V=30.0 PL=1
MOVL C01005 V=130.0 PL=1
MOVL C01006 V=130.0 PL=1
MOVL C01007 V=20.0 PL=1
MOVL C01008 V=130.0 PL=1
MOVL C01009 V=130.0 PL=1
MOVL C01010 V=60.0 PL=1
MOVL C01011 V=60.0 PL=1
MOVL C01012 V=60.0 PL=1
MOVL C01013 V=60.0 PL=1
MOVL C01014 V=130.0 PL=1
MOVL C01015 V=30.0 PL=1
MOVL C01016 V=30.0 PL=1
MOVL C01017 V=30.0 PL=1
MOVL C01018 V=30.0 PL=1
MOVL C01019 V=30.0 PL=1
MOVL C01020 V=30.0 PL=1
MOVL C01021 V=30.0 PL=1
MOVL C01022 V=30.0 PL=1
MOVL C01023 V=130.0 PL=1
MOVL C01024 V=130.0 PL=1
MOVL C01025 V=20.0 PL=1
MOVL C01026 V=130.0 PL=1
MOVL C01027 V=130.0 PL=1
MOVL C01028 V=60.0 PL=1
MOVL C01029 V=60.0 PL=1
MOVL C01030 V=60.0 PL=1
MOVL C01031 V=60.0 PL=1
MOVL C01032 V=130.0 PL=1
MOVL C01033 V=30.0 PL=1
MOVL C01034 V=30.0 PL=1
MOVL C01035 V=30.0 PL=1
MOVL C01036 V=30.0 PL=1
MOVL C01037 V=30.0 PL=1
MOVL C01038 V=30.0 PL=1
MOVL C01039 V=30.0 PL=1
MOVL C01040 V=30.0 PL=1
MOVL C01041 V=130.0 PL=1
MOVL C01042 V=130.0 PL=1
MOVL C01043 V=20.0 PL=1
MOVL C01044 V=130.0 PL=1
MOVL C01045 V=130.0 PL=1
MOVL C01046 V=60.0 PL=1
MOVL C01047 V=60.0 PL=1
MOVL C01048 V=60.0 PL=1
MOVL C01049 V=60.0 PL=1
MOVL C01050 V=130.0 PL=1
MOVL C01051 V=30.0 PL=1
MOVL C01052 V=30.0 PL=1
MOVL C01053 V=30.0 PL=1
MOVL C01054 V=30.0 PL=1
MOVL C01055 V=30.0 PL=1
MOVL C01056 V=30.0 PL=1
MOVL C01057 V=30.0 PL=1
MOVL C01058 V=30.0 PL=1
MOVL C01059 V=130.0 PL=1
MOVL C01060 V=130.0 PL=1
MOVL C01061 V=20.0 PL=1
MOVL C01062 V=130.0 PL=1
MOVL C01063 V=130.0 PL=1
MOVL C01064 V=60.0 PL=1
MOVL C01065 V=60.0 PL=1
MOVL C01066 V=60.0 PL=1
MOVL C01067 V=60.0 PL=1
MOVL C01068 V=130.0 PL=1
MOVL C01069 V=30.0 PL=1
MOVL C01070 V=30.0 PL=1
MOVL C01071 V=30.0 PL=1
MOVL C01072 V=30.0 PL=1
MOVL C01073 V=30.0 PL=1
MOVL C01074 V=30.0 PL=1
MOVL C01075 V=30.0 PL=1
MOVL C01076 V=30.0 PL=1
MOVL C01077 V=130.0 PL=1
MOVL C01078 V=130.0 PL=1
MOVL C01079 V=20.0 PL=1
MOVL C01080 V=130.0 PL=1
MOVL C01081 V=130.0 PL=1
MOVL C01082 V=60.0 PL=1
MOVL C01083 V=60.0 PL=1
MOVL C01084 V=60.0 PL=1
MOVL C01085 V=60.0 PL=1
MOVL C01086 V=130.0 PL=1
MOVL C01087 V=30.0 PL=1
MOVL C01088 V=30.0 PL=1
MOVL C01089 V=30.0 PL=1
MOVL C01090 V=30.0 PL=1
MOVL C01091 V=30.0 PL=1
MOVL C01092 V=30.0 PL=1
MOVL C01093 V=30.0 PL=1
MOVL C01094 V=30.0 PL=1
MOVL C01095 V=130.0 PL=1
MOVL C01096 V=130.0 PL=1
MOVL C01097 V=20.0 PL=1
MOVL C01098 V=130.0 PL=1
MOVL C01099 V=130.0 PL=1
MOVL C01100 V=60.0 PL=1
MOVL C01101 V=60.0 PL=1
MOVL C01102 V=60.0 PL=1
END
